LIN {X 0,Y 590.51,Z 609.214,A -85,B 0,C 180,E1 25169.414,E2 25169.414} C_VEL
LIN {X 0,Y 592.528,Z 625.3,A -85,B 0,C 180,E1 25167.889,E2 25167.889} C_VEL
LIN {X 0,Y 596.332,Z 639.507,A -85,B 0,C 180,E1 25166.405,E2 25166.405} C_VEL
LIN {X 0,Y 601.555,Z 651.727,A -85,B 0,C 180,E1 25165.009,E2 25165.009} C_VEL
LIN {X 0,Y 609.366,Z 664.255,A -85,B 0,C 180,E1 25163.442,E2 25163.442} C_VEL
LIN {X 0,Y 618.653,Z 674.701,A -85,B 0,C 180,E1 25161.991,E2 25161.991} C_VEL
LIN {X 0,Y 629.151,Z 683.449,A -85,B 0,C 180,E1 25160.645,E2 25160.645} C_VEL
LIN {X 0,Y 642.075,Z 691.353,A -85,B 0,C 180,E1 25159.269,E2 25159.269} C_VEL
LIN {X 0,Y 642.773,Z 691.86,A -85,B 0,C 180,E1 25159.192,E2 25159.192} C_VEL
LIN {X 0,Y 632.79,Z 705.423,A -85,B 0,C 180,E1 25158.911,E2 25158.911} C_VEL
LIN {X 0,Y 627.199,Z 713.768,A -85,B 0,C 180,E1 25158.699,E2 25158.699} C_VEL
LIN {X 0,Y 617.726,Z 726.944,A -85,B 0,C 180,E1 25158.399,E2 25158.399} C_VEL
LIN {X 0,Y 610.205,Z 739.734,A -85,B 0,C 180,E1 25157.994,E2 25157.994} C_VEL
LIN {X 0,Y 606.308,Z 747.166,A -85,B 0,C 180,E1 25157.757,E2 25157.757} C_VEL
LIN {X 0,Y 604.005,Z 763.89,A -85,B 0,C 180,E1 25157.714,E2 25157.714} C_VEL
LIN {X 0,Y 603.207,Z 776.285,A -85,B 0,C 180,E1 25157.587,E2 25157.587} C_VEL
LIN {X 0,Y 601.713,Z 819.453,A -85,B 0,C 180,E1 25156.959,E2 25156.959} C_VEL
LIN {X 0,Y 599.605,Z 849.263,A -85,B 0,C 180,E1 25156.4,E2 25156.4} C_VEL
LIN {X 0,Y 597.26,Z 876.114,A -85,B 0,C 180,E1 25155.731,E2 25155.731} C_VEL
LIN {X 0,Y 594.587,Z 902.786,A -85,B 0,C 180,E1 25154.898,E2 25154.898} C_VEL
LIN {X 0,Y 591.585,Z 928.736,A -85,B 0,C 180,E1 25153.901,E2 25153.901} C_VEL
LIN {X 0,Y 588.504,Z 952.603,A -85,B 0,C 180,E1 25152.811,E2 25152.811} C_VEL
LIN {X 0,Y 584.931,Z 977.211,A -85,B 0,C 180,E1 25151.481,E2 25151.481} C_VEL
LIN {X 0,Y 581.177,Z 1000.865,A -85,B 0,C 180,E1 25149.983,E2 25149.983} C_VEL
LIN {X 0,Y 577.362,Z 1023.647,A -85,B 0,C 180,E1 25148.313,E2 25148.313} C_VEL
LIN {X 0,Y 573.393,Z 1045.93,A -85,B 0,C 180,E1 25146.423,E2 25146.423} C_VEL
LIN {X 0,Y 569.931,Z 1065.063,A -85,B 0,C 180,E1 25144.577,E2 25144.577} C_VEL
LIN {X 0,Y 566.236,Z 1085.757,A -85,B 0,C 180,E1 25142.312,E2 25142.312} C_VEL
LIN {X 0,Y 563.29,Z 1102.922,A -85,B 0,C 180,E1 25140.177,E2 25140.177} C_VEL
LIN {X 0,Y 560.401,Z 1120.145,A -85,B 0,C 180,E1 25137.75,E2 25137.75} C_VEL
LIN {X 0,Y 558.227,Z 1134.517,A -85,B 0,C 180,E1 25135.458,E2 25135.458} C_VEL
LIN {X 0,Y 556.22,Z 1148.88,A -85,B 0,C 180,E1 25132.847,E2 25132.847} C_VEL
LIN {X 0,Y 554.619,Z 1162.074,A -85,B 0,C 180,E1 25130.068,E2 25130.068} C_VEL
LIN {X 0,Y 553.529,Z 1172.793,A -85,B 0,C 180,E1 25127.448,E2 25127.448} C_VEL
LIN {X 0,Y 552.746,Z 1182.624,A -85,B 0,C 180,E1 25124.581,E2 25124.581} C_VEL
LIN {X 0,Y 552.293,Z 1190.071,A -85,B 0,C 180,E1 25121.909,E2 25121.909} C_VEL
LIN {X 0,Y 552.049,Z 1196.15,A -85,B 0,C 180,E1 25119.17,E2 25119.17} C_VEL
LIN {X 0,Y 551.953,Z 1200.501,A -85,B 0,C 180,E1 25116.552,E2 25116.552} C_VEL
LIN {X 0,Y 551.914,Z 1203.328,A -85,B 0,C 180,E1 25113.946,E2 25113.946} C_VEL
LIN {X 0,Y 551.916,Z 1204.787,A -85,B 0,C 180,E1 25111.244,E2 25111.244} C_VEL
LIN {X 0,Y 551.916,Z 1204.786,A -85,B 0,C 180,E1 25108.753,E2 25108.753} C_VEL
LIN {X 0,Y 551.914,Z 1203.326,A -85,B 0,C 180,E1 25106.051,E2 25106.051} C_VEL
LIN {X 0,Y 551.951,Z 1200.497,A -85,B 0,C 180,E1 25103.445,E2 25103.445} C_VEL
LIN {X 0,Y 552.051,Z 1196.087,A -85,B 0,C 180,E1 25100.796,E2 25100.796} C_VEL
LIN {X 0,Y 552.293,Z 1190.065,A -85,B 0,C 180,E1 25098.088,E2 25098.088} C_VEL
LIN {X 0,Y 552.746,Z 1182.623,A -85,B 0,C 180,E1 25095.419,E2 25095.419} C_VEL
LIN {X 0,Y 553.529,Z 1172.783,A -85,B 0,C 180,E1 25092.55,E2 25092.55} C_VEL
LIN {X 0,Y 554.62,Z 1162.073,A -85,B 0,C 180,E1 25089.932,E2 25089.932} C_VEL
LIN {X 0,Y 556.222,Z 1148.866,A -85,B 0,C 180,E1 25087.151,E2 25087.151} C_VEL
LIN {X 0,Y 558.249,Z 1134.381,A -85,B 0,C 180,E1 25084.519,E2 25084.519} C_VEL
LIN {X 0,Y 560.406,Z 1120.11,A -85,B 0,C 180,E1 25082.245,E2 25082.245} C_VEL
LIN {X 0,Y 563.403,Z 1102.225,A -85,B 0,C 180,E1 25079.733,E2 25079.733} C_VEL
LIN {X 0,Y 566.285,Z 1085.478,A -85,B 0,C 180,E1 25077.655,E2 25077.655} C_VEL
LIN {X 0,Y 569.935,Z 1065.037,A -85,B 0,C 180,E1 25075.42,E2 25075.42} C_VEL
LIN {X 0,Y 573.399,Z 1045.901,A -85,B 0,C 180,E1 25073.575,E2 25073.575} C_VEL
LIN {X 0,Y 577.128,Z 1024.944,A -85,B 0,C 180,E1 25071.792,E2 25071.792} C_VEL
LIN {X 0,Y 580.932,Z 1002.513,A -85,B 0,C 180,E1 25070.129,E2 25070.129} C_VEL
LIN {X 0,Y 584.659,Z 978.962,A -85,B 0,C 180,E1 25068.623,E2 25068.623} C_VEL
LIN {X 0,Y 588.218,Z 954.716,A -85,B 0,C 180,E1 25067.293,E2 25067.293} C_VEL
LIN {X 0,Y 591.704,Z 928.188,A -85,B 0,C 180,E1 25066.07,E2 25066.07} C_VEL
LIN {X 0,Y 594.755,Z 901.513,A -85,B 0,C 180,E1 25065.055,E2 25065.055} C_VEL
LIN {X 0,Y 597.525,Z 873.698,A -85,B 0,C 180,E1 25064.197,E2 25064.197} C_VEL
LIN {X 0,Y 600.006,Z 844.404,A -85,B 0,C 180,E1 25063.494,E2 25063.494} C_VEL
LIN {X 0,Y 602.162,Z 810.979,A -85,B 0,C 180,E1 25062.904,E2 25062.904} C_VEL
LIN {X 0,Y 604.764,Z 734.901,A -85,B 0,C 180,E1 25061.837,E2 25061.837} C_VEL
LIN {X 0,Y 611.43,Z 660.897,A -85,B 0,C 180,E1 25060.584,E2 25060.584} C_VEL
LIN {X 0,Y 612.883,Z 645.219,A -85,B 0,C 180,E1 25060.323,E2 25060.323} C_VEL
LIN {X 0,Y 616.334,Z 610.333,A -85,B 0,C 180,E1 25059.764,E2 25059.764} C_VEL
LIN {X 0,Y 617.889,Z 595.942,A -85,B 0,C 180,E1 25059.548,E2 25059.548} C_VEL
LIN {X 0,Y 620.532,Z 567.007,A -85,B 0,C 180,E1 25059.061,E2 25059.061} C_VEL
LIN {X 0,Y 624,Z 538.188,A -85,B 0,C 180,E1 25058.666,E2 25058.666} C_VEL
LIN {X 0,Y 626.222,Z 512.687,A -85,B 0,C 180,E1 25058.225,E2 25058.225} C_VEL
LIN {X 0,Y 630.739,Z 478.238,A -85,B 0,C 180,E1 25057.795,E2 25057.795} C_VEL
LIN {X 0,Y 632.724,Z 453.547,A -85,B 0,C 180,E1 25057.35,E2 25057.35} C_VEL
LIN {X 0,Y 633.686,Z 444.389,A -85,B 0,C 180,E1 25057.21,E2 25057.21} C_VEL
LIN {X 0,Y 625.904,Z 434.82,A -85,B 0,C 180,E1 25056.064,E2 25056.064} C_VEL
LIN {X 0,Y 610.871,Z 411.674,A -85,B 0,C 180,E1 25053.534,E2 25053.534} C_VEL
LIN {X 0,Y 599.2,Z 394.973,A -85,B 0,C 180,E1 25051.403,E2 25051.403} C_VEL
LIN {X 0,Y 589.319,Z 381.338,A -85,B 0,C 180,E1 25049.447,E2 25049.447} C_VEL
LIN {X 0,Y 584.227,Z 374.732,A -85,B 0,C 180,E1 25048.383,E2 25048.383} C_VEL
LIN {X 0,Y 581.035,Z 370.541,A -85,B 0,C 180,E1 25047.687,E2 25047.687} C_VEL
LIN {X 0,Y 576.918,Z 365.165,A -85,B 0,C 180,E1 25046.756,E2 25046.756} C_VEL
LIN {X 0,Y 573.423,Z 360.486,A -85,B 0,C 180,E1 25045.928,E2 25045.928} C_VEL
LIN {X 0,Y 569.377,Z 355.739,A -85,B 0,C 180,E1 25044.955,E2 25044.955} C_VEL
LIN {X 0,Y 568.216,Z 353.937,A -85,B 0,C 180,E1 25044.649,E2 25044.649} C_VEL
LIN {X 0,Y 565.016,Z 350.609,A -85,B 0,C 180,E1 25043.852,E2 25043.852} C_VEL
LIN {X 0,Y 563.518,Z 347.975,A -85,B 0,C 180,E1 25043.42,E2 25043.42} C_VEL
LIN {X 0,Y 560.374,Z 345.311,A -85,B 0,C 180,E1 25042.614,E2 25042.614} C_VEL
LIN {X 0,Y 558.326,Z 341.668,A -85,B 0,C 180,E1 25041.981,E2 25041.981} C_VEL
LIN {X 0,Y 555.306,Z 339.437,A -85,B 0,C 180,E1 25041.163,E2 25041.163} C_VEL
LIN {X 0,Y 553.735,Z 336.439,A -85,B 0,C 180,E1 25040.631,E2 25040.631} C_VEL
LIN {X 0,Y 553.497,Z 335.263,A -85,B 0,C 180,E1 25040.488,E2 25040.488} C_VEL
LIN {X 0,Y 553.496,Z 335.262,A -85,B 0,C 180,E1 25037.017,E2 25037.017} C_VEL
LIN {X 0,Y 553.524,Z 335.519,A -85,B 0,C 180,E1 25035.601,E2 25035.601} C_VEL
LIN {X 0,Y 560.446,Z 355.632,A -85,B 0,C 180,E1 25034.584,E2 25034.584} C_VEL
LIN {X 0,Y 560.203,Z 434.439,A -85,B 0,C 180,E1 25031.766,E2 25031.766} C_VEL
LIN {X 0,Y 560.354,Z 519.456,A -85,B 0,C 180,E1 25028.569,E2 25028.569} C_VEL
LIN {X 0,Y 560.071,Z 596.427,A -85,B 0,C 180,E1 25025.584,E2 25025.584} C_VEL
LIN {X 0,Y 559.404,Z 672.282,A -85,B 0,C 180,E1 25022.561,E2 25022.561} C_VEL
LIN {X 0,Y 558.433,Z 749.146,A -85,B 0,C 180,E1 25019.436,E2 25019.436} C_VEL
LIN {X 0,Y 557.327,Z 828.653,A -85,B 0,C 180,E1 25016.142,E2 25016.142} C_VEL
LIN {X 0,Y 556.701,Z 851.757,A -85,B 0,C 180,E1 25015.186,E2 25015.186} C_VEL
LIN {X 0,Y 556.119,Z 860.24,A -85,B 0,C 180,E1 25014.87,E2 25014.87} C_VEL
LIN {X 0,Y 555.338,Z 973.856,A -85,B 0,C 180,E1 25013.286,E2 25013.286} C_VEL
LIN {X 0,Y 555.38,Z 986.399,A -85,B 0,C 180,E1 25012.978,E2 25012.978} C_VEL
LIN {X 0,Y 555.343,Z 998.353,A -85,B 0,C 180,E1 25012.551,E2 25012.551} C_VEL
LIN {X 0,Y 555.203,Z 1011.407,A -85,B 0,C 180,E1 25011.925,E2 25011.925} C_VEL
LIN {X 0,Y 554.96,Z 1023.564,A -85,B 0,C 180,E1 25011.132,E2 25011.132} C_VEL
LIN {X 0,Y 554.721,Z 1033.15,A -85,B 0,C 180,E1 25010.35,E2 25010.35} C_VEL
LIN {X 0,Y 554.462,Z 1041.636,A -85,B 0,C 180,E1 25009.506,E2 25009.506} C_VEL
LIN {X 0,Y 554.197,Z 1049.49,A -85,B 0,C 180,E1 25008.553,E2 25008.553} C_VEL
LIN {X 0,Y 553.925,Z 1057.258,A -85,B 0,C 180,E1 25007.384,E2 25007.384} C_VEL
LIN {X 0,Y 553.645,Z 1064.108,A -85,B 0,C 180,E1 25005.995,E2 25005.995} C_VEL
LIN {X 0,Y 553.48,Z 1068.39,A -85,B 0,C 180,E1 25004.814,E2 25004.814} C_VEL
LIN {X 0,Y 553.352,Z 1071.423,A -85,B 0,C 180,E1 25003.627,E2 25003.627} C_VEL
LIN {X 0,Y 553.276,Z 1073.272,A -85,B 0,C 180,E1 25002.434,E2 25002.434} C_VEL
LIN {X 0,Y 553.227,Z 1074.038,A -85,B 0,C 180,E1 25001.014,E2 25001.014} C_VEL
LIN {X 0,Y 553.232,Z 1072.866,A -85,B 0,C 180,E1 24999.426,E2 24999.426} C_VEL
LIN {X 0,Y 553.274,Z 1070.476,A -85,B 0,C 180,E1 24998.143,E2 24998.143} C_VEL
LIN {X 0,Y 553.376,Z 1066.816,A -85,B 0,C 180,E1 24996.884,E2 24996.884} C_VEL
LIN {X 0,Y 553.578,Z 1060.937,A -85,B 0,C 180,E1 24995.453,E2 24995.453} C_VEL
LIN {X 0,Y 553.81,Z 1053.905,A -85,B 0,C 180,E1 24994.207,E2 24994.207} C_VEL
LIN {X 0,Y 554.066,Z 1046.433,A -85,B 0,C 180,E1 24993.151,E2 24993.151} C_VEL
LIN {X 0,Y 554.352,Z 1037.727,A -85,B 0,C 180,E1 24992.15,E2 24992.15} C_VEL
LIN {X 0,Y 554.704,Z 1026.532,A -85,B 0,C 180,E1 24991.113,E2 24991.113} C_VEL
LIN {X 0,Y 554.983,Z 1014.283,A -85,B 0,C 180,E1 24990.241,E2 24990.241} C_VEL
LIN {X 0,Y 555.2,Z 1003.236,A -85,B 0,C 180,E1 24989.617,E2 24989.617} C_VEL
LIN {X 0,Y 555.368,Z 990.76,A -85,B 0,C 180,E1 24989.071,E2 24989.071} C_VEL
LIN {X 0,Y 555.439,Z 974.896,A -85,B 0,C 180,E1 24988.598,E2 24988.598} C_VEL
LIN {X 0,Y 555.398,Z 958.822,A -85,B 0,C 180,E1 24988.323,E2 24988.323} C_VEL
LIN {X 0,Y 556.342,Z 853.596,A -85,B 0,C 180,E1 24986.88,E2 24986.88} C_VEL
LIN {X 0,Y 557.037,Z 837.818,A -85,B 0,C 180,E1 24986.212,E2 24986.212} C_VEL
LIN {X 0,Y 558.557,Z 756.681,A -85,B 0,C 180,E1 24982.702,E2 24982.702} C_VEL
LIN {X 0,Y 558.996,Z 735.045,A -85,B 0,C 180,E1 24981.765,E2 24981.765} C_VEL
LIN {X 0,Y 559.725,Z 732.326,A -85,B 0,C 180,E1 24981.556,E2 24981.556} C_VEL
LIN {X 0,Y 561.703,Z 730.328,A -85,B 0,C 180,E1 24981.216,E2 24981.216} C_VEL
LIN {X 0,Y 566.453,Z 728.934,A -85,B 0,C 180,E1 24980.588,E2 24980.588} C_VEL
LIN {X 0,Y 571.435,Z 727.549,A -85,B 0,C 180,E1 24980.042,E2 24980.042} C_VEL
LIN {X 0,Y 572.537,Z 726.951,A -85,B 0,C 180,E1 24979.933,E2 24979.933} C_VEL
LIN {X 0,Y 577.099,Z 723.151,A -85,B 0,C 180,E1 24979.527,E2 24979.527} C_VEL
LIN {X 0,Y 582.053,Z 717.036,A -85,B 0,C 180,E1 24979.15,E2 24979.15} C_VEL
LIN {X 0,Y 587.21,Z 712.981,A -85,B 0,C 180,E1 24978.713,E2 24978.713} C_VEL
LIN {X 0,Y 593.112,Z 706.301,A -85,B 0,C 180,E1 24978.28,E2 24978.28} C_VEL
LIN {X 0,Y 594.096,Z 705.686,A -85,B 0,C 180,E1 24978.198,E2 24978.198} C_VEL
LIN {X 0,Y 589.64,Z 797.135,A -85,B 0,C 180,E1 24976.661,E2 24976.661} C_VEL
LIN {X 0,Y 588.016,Z 826.067,A -85,B 0,C 180,E1 24976.11,E2 24976.11} C_VEL
LIN {X 0,Y 585.936,Z 855.454,A -85,B 0,C 180,E1 24975.37,E2 24975.37} C_VEL
LIN {X 0,Y 583.804,Z 880.901,A -85,B 0,C 180,E1 24974.562,E2 24974.562} C_VEL
LIN {X 0,Y 581.521,Z 904.72,A -85,B 0,C 180,E1 24973.659,E2 24973.659} C_VEL
LIN {X 0,Y 578.69,Z 930.131,A -85,B 0,C 180,E1 24972.501,E2 24972.501} C_VEL
LIN {X 0,Y 575.93,Z 952.54,A -85,B 0,C 180,E1 24971.317,E2 24971.317} C_VEL
LIN {X 0,Y 572.684,Z 976.437,A -85,B 0,C 180,E1 24969.85,E2 24969.85} C_VEL
LIN {X 0,Y 568.97,Z 1000.766,A -85,B 0,C 180,E1 24968.086,E2 24968.086} C_VEL
LIN {X 0,Y 565.934,Z 1019.321,A -85,B 0,C 180,E1 24966.543,E2 24966.543} C_VEL
LIN {X 0,Y 563.293,Z 1033.801,A -85,B 0,C 180,E1 24965.142,E2 24965.142} C_VEL
LIN {X 0,Y 560.146,Z 1050.417,A -85,B 0,C 180,E1 24963.342,E2 24963.342} C_VEL
LIN {X 0,Y 557.391,Z 1065.236,A -85,B 0,C 180,E1 24961.56,E2 24961.56} C_VEL
LIN {X 0,Y 554.87,Z 1079.174,A -85,B 0,C 180,E1 24959.706,E2 24959.706} C_VEL
LIN {X 0,Y 552.605,Z 1092.304,A -85,B 0,C 180,E1 24957.772,E2 24957.772} C_VEL
LIN {X 0,Y 550.606,Z 1104.824,A -85,B 0,C 180,E1 24955.724,E2 24955.724} C_VEL
LIN {X 0,Y 548.637,Z 1118.142,A -85,B 0,C 180,E1 24953.286,E2 24953.286} C_VEL
LIN {X 0,Y 546.891,Z 1131.542,A -85,B 0,C 180,E1 24950.44,E2 24950.44} C_VEL
LIN {X 0,Y 545.8,Z 1141.259,A -85,B 0,C 180,E1 24948.048,E2 24948.048} C_VEL
LIN {X 0,Y 545.07,Z 1148.997,A -85,B 0,C 180,E1 24945.864,E2 24945.864} C_VEL
LIN {X 0,Y 544.565,Z 1155.927,A -85,B 0,C 180,E1 24943.594,E2 24943.594} C_VEL
LIN {X 0,Y 544.215,Z 1161.96,A -85,B 0,C 180,E1 24941.232,E2 24941.232} C_VEL
LIN {X 0,Y 544.045,Z 1166.607,A -85,B 0,C 180,E1 24938.989,E2 24938.989} C_VEL
LIN {X 0,Y 543.953,Z 1170.204,A -85,B 0,C 180,E1 24936.757,E2 24936.757} C_VEL
LIN {X 0,Y 543.916,Z 1172.778,A -85,B 0,C 180,E1 24934.535,E2 24934.535} C_VEL
LIN {X 0,Y 543.908,Z 1174.344,A -85,B 0,C 180,E1 24932.319,E2 24932.319} C_VEL
LIN {X 0,Y 543.907,Z 1174.912,A -85,B 0,C 180,E1 24929.896,E2 24929.896} C_VEL
LIN {X 0,Y 543.907,Z 1174.289,A -85,B 0,C 180,E1 24927.473,E2 24927.473} C_VEL
LIN {X 0,Y 543.92,Z 1172.538,A -85,B 0,C 180,E1 24925.114,E2 24925.114} C_VEL
LIN {X 0,Y 543.973,Z 1169.598,A -85,B 0,C 180,E1 24922.715,E2 24922.715} C_VEL
LIN {X 0,Y 544.113,Z 1164.806,A -85,B 0,C 180,E1 24919.947,E2 24919.947} C_VEL
LIN {X 0,Y 544.467,Z 1157.685,A -85,B 0,C 180,E1 24916.947,E2 24916.947} C_VEL
LIN {X 0,Y 544.968,Z 1150.356,A -85,B 0,C 180,E1 24914.464,E2 24914.464} C_VEL
LIN {X 0,Y 545.68,Z 1142.458,A -85,B 0,C 180,E1 24912.183,E2 24912.183} C_VEL
LIN {X 0,Y 546.618,Z 1133.78,A -85,B 0,C 180,E1 24909.999,E2 24909.999} C_VEL
LIN {X 0,Y 547.759,Z 1124.416,A -85,B 0,C 180,E1 24907.913,E2 24907.913} C_VEL
LIN {X 0,Y 549.227,Z 1113.891,A -85,B 0,C 180,E1 24905.821,E2 24905.821} C_VEL
LIN {X 0,Y 551.035,Z 1101.917,A -85,B 0,C 180,E1 24903.689,E2 24903.689} C_VEL
LIN {X 0,Y 553.601,Z 1086.776,A -85,B 0,C 180,E1 24901.288,E2 24901.288} C_VEL
LIN {X 0,Y 556.821,Z 1068.311,A -85,B 0,C 180,E1 24898.739,E2 24898.739} C_VEL
LIN {X 0,Y 559.75,Z 1052.486,A -85,B 0,C 180,E1 24896.806,E2 24896.806} C_VEL
LIN {X 0,Y 562.67,Z 1036.971,A -85,B 0,C 180,E1 24895.098,E2 24895.098} C_VEL
LIN {X 0,Y 565.344,Z 1022.647,A -85,B 0,C 180,E1 24893.668,E2 24893.668} C_VEL
LIN {X 0,Y 567.988,Z 1006.559,A -85,B 0,C 180,E1 24892.287,E2 24892.287} C_VEL
LIN {X 0,Y 571.311,Z 985.32,A -85,B 0,C 180,E1 24890.676,E2 24890.676} C_VEL
LIN {X 0,Y 574.184,Z 965.577,A -85,B 0,C 180,E1 24889.364,E2 24889.364} C_VEL
LIN {X 0,Y 576.941,Z 944.473,A -85,B 0,C 180,E1 24888.148,E2 24888.148} C_VEL
LIN {X 0,Y 579.829,Z 920.099,A -85,B 0,C 180,E1 24886.933,E2 24886.933} C_VEL
LIN {X 0,Y 582.213,Z 897.637,A -85,B 0,C 180,E1 24885.969,E2 24885.969} C_VEL
LIN {X 0,Y 584.057,Z 877.701,A -85,B 0,C 180,E1 24885.242,E2 24885.242} C_VEL
LIN {X 0,Y 586.31,Z 850.909,A -85,B 0,C 180,E1 24884.413,E2 24884.413} C_VEL
LIN {X 0,Y 587.914,Z 826.678,A -85,B 0,C 180,E1 24883.823,E2 24883.823} C_VEL
LIN {X 0,Y 589.099,Z 806.755,A -85,B 0,C 180,E1 24883.424,E2 24883.424} C_VEL
LIN {X 0,Y 595.542,Z 680.019,A -85,B 0,C 180,E1 24881.271,E2 24881.271} C_VEL
LIN {X 0,Y 603.788,Z 534.875,A -85,B 0,C 180,E1 24878.84,E2 24878.84} C_VEL
LIN {X 0,Y 608.499,Z 434.897,A -85,B 0,C 180,E1 24877.284,E2 24877.284} C_VEL
LIN {X 0,Y 608.958,Z 420.597,A -85,B 0,C 180,E1 24877.057,E2 24877.057} C_VEL
LIN {X 0,Y 597.614,Z 409.55,A -85,B 0,C 180,E1 24875.344,E2 24875.344} C_VEL
LIN {X 0,Y 588.958,Z 401.686,A -85,B 0,C 180,E1 24873.956,E2 24873.956} C_VEL
LIN {X 0,Y 582.445,Z 395.957,A -85,B 0,C 180,E1 24872.853,E2 24872.853} C_VEL
LIN {X 0,Y 579.818,Z 393.63,A -85,B 0,C 180,E1 24872.369,E2 24872.369} C_VEL
LIN {X 0,Y 578.408,Z 390.814,A -85,B 0,C 180,E1 24871.355,E2 24871.355} C_VEL
LIN {X 0,Y 575.887,Z 386.066,A -85,B 0,C 180,E1 24869.43,E2 24869.43} C_VEL
LIN {X 0,Y 573.641,Z 381.867,A -85,B 0,C 180,E1 24867.479,E2 24867.479} C_VEL
LIN {X 0,Y 570.817,Z 376.935,A -85,B 0,C 180,E1 24864.621,E2 24864.621} C_VEL
LIN {X 0,Y 570.206,Z 375.881,A -85,B 0,C 180,E1 24863.896,E2 24863.896} C_VEL
LIN {X 0,Y 567.555,Z 370.875,A -85,B 0,C 180,E1 24859.449,E2 24859.449} C_VEL
LIN {X 0,Y 566.073,Z 369.458,A -85,B 0,C 180,E1 24854.84,E2 24854.84} C_VEL
LIN {X 0,Y 566.639,Z 370.081,A -85,B 0,C 180,E1 24850.781,E2 24850.781} C_VEL
LIN {X 0,Y 567.835,Z 371.39,A -85,B 0,C 180,E1 24848.28,E2 24848.28} C_VEL
LIN {X 0,Y 570.94,Z 376.86,A -85,B 0,C 180,E1 24843.715,E2 24843.715} C_VEL
LIN {X 0,Y 573.241,Z 381.117,A -85,B 0,C 180,E1 24841.299,E2 24841.299} C_VEL
LIN {X 0,Y 573.954,Z 382.347,A -85,B 0,C 180,E1 24840.664,E2 24840.664} C_VEL
LIN {X 0,Y 576.229,Z 386.32,A -85,B 0,C 180,E1 24838.807,E2 24838.807} C_VEL
LIN {X 0,Y 579.608,Z 392.611,A -85,B 0,C 180,E1 24836.34,E2 24836.34} C_VEL
LIN {X 0,Y 582.344,Z 397.71,A -85,B 0,C 180,E1 24834.581,E2 24834.581} C_VEL
LIN {X 0,Y 584.961,Z 402.676,A -85,B 0,C 180,E1 24833.029,E2 24833.029} C_VEL
LIN {X 0,Y 587.586,Z 407.673,A -85,B 0,C 180,E1 24831.585,E2 24831.585} C_VEL
LIN {X 0,Y 591.706,Z 415.65,A -85,B 0,C 180,E1 24829.484,E2 24829.484} C_VEL
LIN {X 0,Y 597.53,Z 427.473,A -85,B 0,C 180,E1 24826.747,E2 24826.747} C_VEL
LIN {X 0,Y 603.495,Z 440.421,A -85,B 0,C 180,E1 24824.135,E2 24824.135} C_VEL
LIN {X 0,Y 604.72,Z 443.335,A -85,B 0,C 180,E1 24823.601,E2 24823.601} C_VEL
LIN {X 0,Y 599.356,Z 478.045,A -85,B 0,C 180,E1 24820.61,E2 24820.61} C_VEL
LIN {X 0,Y 594.302,Z 512.72,A -85,B 0,C 180,E1 24817.756,E2 24817.756} C_VEL
LIN {X 0,Y 589.378,Z 549.232,A -85,B 0,C 180,E1 24814.851,E2 24814.851} C_VEL
LIN {X 0,Y 584.185,Z 594.684,A -85,B 0,C 180,E1 24811.308,E2 24811.308} C_VEL
LIN {X 0,Y 584.176,Z 612.88,A -85,B 0,C 180,E1 24809.73,E2 24809.73} C_VEL
LIN {X 0,Y 586.102,Z 628.98,A -85,B 0,C 180,E1 24808.186,E2 24808.186} C_VEL
LIN {X 0,Y 589.787,Z 643.265,A -85,B 0,C 180,E1 24806.681,E2 24806.681} C_VEL
LIN {X 0,Y 594.874,Z 655.617,A -85,B 0,C 180,E1 24805.263,E2 24805.263} C_VEL
LIN {X 0,Y 602.522,Z 668.326,A -85,B 0,C 180,E1 24803.669,E2 24803.669} C_VEL
LIN {X 0,Y 611.632,Z 679.01,A -85,B 0,C 180,E1 24802.19,E2 24802.19} C_VEL
LIN {X 0,Y 622.56,Z 688.475,A -85,B 0,C 180,E1 24800.743,E2 24800.743} C_VEL
LIN {X 0,Y 632.882,Z 695.437,A -85,B 0,C 180,E1 24799.579,E2 24799.579} C_VEL
LIN {X 0,Y 624.075,Z 708.29,A -85,B 0,C 180,E1 24799.271,E2 24799.271} C_VEL
LIN {X 0,Y 612.294,Z 724.665,A -85,B 0,C 180,E1 24798.904,E2 24798.904} C_VEL
LIN {X 0,Y 604.358,Z 738.022,A -85,B 0,C 180,E1 24798.486,E2 24798.486} C_VEL
LIN {X 0,Y 601.573,Z 743.536,A -85,B 0,C 180,E1 24798.316,E2 24798.316} C_VEL
LIN {X 0,Y 599.265,Z 758.516,A -85,B 0,C 180,E1 24798.304,E2 24798.304} C_VEL
LIN {X 0,Y 597.904,Z 773.102,A -85,B 0,C 180,E1 24798.198,E2 24798.198} C_VEL
LIN {X 0,Y 596.316,Z 817.198,A -85,B 0,C 180,E1 24797.553,E2 24797.553} C_VEL
LIN {X 0,Y 594.025,Z 848.758,A -85,B 0,C 180,E1 24796.963,E2 24796.963} C_VEL
LIN {X 0,Y 591.422,Z 877.702,A -85,B 0,C 180,E1 24796.238,E2 24796.238} C_VEL
LIN {X 0,Y 588.576,Z 904.677,A -85,B 0,C 180,E1 24795.38,E2 24795.38} C_VEL
LIN {X 0,Y 585.764,Z 927.976,A -85,B 0,C 180,E1 24794.478,E2 24794.478} C_VEL
LIN {X 0,Y 582.666,Z 951.398,A -85,B 0,C 180,E1 24793.413,E2 24793.413} C_VEL
LIN {X 0,Y 579.101,Z 975.478,A -85,B 0,C 180,E1 24792.126,E2 24792.126} C_VEL
LIN {X 0,Y 575.44,Z 997.395,A -85,B 0,C 180,E1 24790.747,E2 24790.747} C_VEL
LIN {X 0,Y 571.21,Z 1021.62,A -85,B 0,C 180,E1 24788.994,E2 24788.994} C_VEL
LIN {X 0,Y 567.046,Z 1044.191,A -85,B 0,C 180,E1 24787.087,E2 24787.087} C_VEL
LIN {X 0,Y 563.262,Z 1063.982,A -85,B 0,C 180,E1 24785.171,E2 24785.171} C_VEL
LIN {X 0,Y 559.56,Z 1083.663,A -85,B 0,C 180,E1 24783.023,E2 24783.023} C_VEL
LIN {X 0,Y 556.432,Z 1100.552,A -85,B 0,C 180,E1 24780.924,E2 24780.924} C_VEL
LIN {X 0,Y 553.386,Z 1117.974,A -85,B 0,C 180,E1 24778.488,E2 24778.488} C_VEL
LIN {X 0,Y 550.857,Z 1133.198,A -85,B 0,C 180,E1 24776.055,E2 24776.055} C_VEL
LIN {X 0,Y 548.685,Z 1147.76,A -85,B 0,C 180,E1 24773.406,E2 24773.406} C_VEL
LIN {X 0,Y 546.969,Z 1160.827,A -85,B 0,C 180,E1 24770.658,E2 24770.658} C_VEL
LIN {X 0,Y 545.788,Z 1171.565,A -85,B 0,C 180,E1 24768.034,E2 24768.034} C_VEL
LIN {X 0,Y 544.936,Z 1180.951,A -85,B 0,C 180,E1 24765.319,E2 24765.319} C_VEL
LIN {X 0,Y 544.375,Z 1188.99,A -85,B 0,C 180,E1 24762.516,E2 24762.516} C_VEL
LIN {X 0,Y 544.095,Z 1195.366,A -85,B 0,C 180,E1 24759.732,E2 24759.732} C_VEL
LIN {X 0,Y 543.965,Z 1199.881,A -85,B 0,C 180,E1 24757.073,E2 24757.073} C_VEL
LIN {X 0,Y 543.92,Z 1203.062,A -85,B 0,C 180,E1 24754.321,E2 24754.321} C_VEL
LIN {X 0,Y 543.908,Z 1204.699,A -85,B 0,C 180,E1 24751.684,E2 24751.684} C_VEL
LIN {X 0,Y 543.907,Z 1204.845,A -85,B 0,C 180,E1 24749.051,E2 24749.051} C_VEL
LIN {X 0,Y 543.913,Z 1203.677,A -85,B 0,C 180,E1 24746.415,E2 24746.415} C_VEL
LIN {X 0,Y 543.945,Z 1201.031,A -85,B 0,C 180,E1 24743.773,E2 24743.773} C_VEL
LIN {X 0,Y 544.038,Z 1196.928,A -85,B 0,C 180,E1 24741.118,E2 24741.118} C_VEL
LIN {X 0,Y 544.258,Z 1191.41,A -85,B 0,C 180,E1 24738.447,E2 24738.447} C_VEL
LIN {X 0,Y 544.712,Z 1183.952,A -85,B 0,C 180,E1 24735.651,E2 24735.651} C_VEL
LIN {X 0,Y 545.491,Z 1174.422,A -85,B 0,C 180,E1 24732.747,E2 24732.747} C_VEL
LIN {X 0,Y 546.638,Z 1163.636,A -85,B 0,C 180,E1 24729.997,E2 24729.997} C_VEL
LIN {X 0,Y 548.163,Z 1151.659,A -85,B 0,C 180,E1 24727.363,E2 24727.363} C_VEL
LIN {X 0,Y 550.326,Z 1136.805,A -85,B 0,C 180,E1 24724.556,E2 24724.556} C_VEL
LIN {X 0,Y 552.742,Z 1121.545,A -85,B 0,C 180,E1 24722.061,E2 24722.061} C_VEL
LIN {X 0,Y 555.728,Z 1104.764,A -85,B 0,C 180,E1 24719.629,E2 24719.629} C_VEL
LIN {X 0,Y 558.943,Z 1086.852,A -85,B 0,C 180,E1 24717.36,E2 24717.36} C_VEL
LIN {X 0,Y 562.586,Z 1067.591,A -85,B 0,C 180,E1 24715.197,E2 24715.197} C_VEL
LIN {X 0,Y 566.606,Z 1046.593,A -85,B 0,C 180,E1 24713.129,E2 24713.129} C_VEL
LIN {X 0,Y 570.212,Z 1027.155,A -85,B 0,C 180,E1 24711.452,E2 24711.452} C_VEL
LIN {X 0,Y 574.41,Z 1003.744,A -85,B 0,C 180,E1 24709.68,E2 24709.68} C_VEL
LIN {X 0,Y 578.265,Z 980.684,A -85,B 0,C 180,E1 24708.181,E2 24708.181} C_VEL
LIN {X 0,Y 582.05,Z 955.634,A -85,B 0,C 180,E1 24706.797,E2 24706.797} C_VEL
LIN {X 0,Y 585.496,Z 930.62,A -85,B 0,C 180,E1 24705.626,E2 24705.626} C_VEL
LIN {X 0,Y 588.686,Z 903.882,A -85,B 0,C 180,E1 24704.59,E2 24704.59} C_VEL
LIN {X 0,Y 591.584,Z 876.02,A -85,B 0,C 180,E1 24703.714,E2 24703.714} C_VEL
LIN {X 0,Y 594.182,Z 846.963,A -85,B 0,C 180,E1 24702.996,E2 24702.996} C_VEL
LIN {X 0,Y 596.465,Z 814.54,A -85,B 0,C 180,E1 24702.403,E2 24702.403} C_VEL
LIN {X 0,Y 598.405,Z 756.727,A -85,B 0,C 180,E1 24701.575,E2 24701.575} C_VEL
LIN {X 0,Y 599.593,Z 730.221,A -85,B 0,C 180,E1 24701.198,E2 24701.198} C_VEL
LIN {X 0,Y 606.118,Z 660.111,A -85,B 0,C 180,E1 24700.016,E2 24700.016} C_VEL
LIN {X 0,Y 607.72,Z 642.456,A -85,B 0,C 180,E1 24699.714,E2 24699.714} C_VEL
LIN {X 0,Y 611.474,Z 606.607,A -85,B 0,C 180,E1 24699.154,E2 24699.154} C_VEL
LIN {X 0,Y 612.598,Z 595.536,A -85,B 0,C 180,E1 24698.977,E2 24698.977} C_VEL
LIN {X 0,Y 615.456,Z 565.573,A -85,B 0,C 180,E1 24698.479,E2 24698.479} C_VEL
LIN {X 0,Y 618.733,Z 538.714,A -85,B 0,C 180,E1 24698.11,E2 24698.11} C_VEL
LIN {X 0,Y 621.076,Z 512.63,A -85,B 0,C 180,E1 24697.661,E2 24697.661} C_VEL
LIN {X 0,Y 625.775,Z 476.02,A -85,B 0,C 180,E1 24697.187,E2 24697.187} C_VEL
LIN {X 0,Y 627.695,Z 453.263,A -85,B 0,C 180,E1 24696.781,E2 24696.781} C_VEL
LIN {X 0,Y 628.114,Z 448.951,A -85,B 0,C 180,E1 24696.71,E2 24696.71} C_VEL
LIN {X 0,Y 620.495,Z 438.824,A -85,B 0,C 180,E1 24695.538,E2 24695.538} C_VEL
LIN {X 0,Y 607.119,Z 417.981,A -85,B 0,C 180,E1 24693.232,E2 24693.232} C_VEL
LIN {X 0,Y 594.255,Z 399.296,A -85,B 0,C 180,E1 24690.821,E2 24690.821} C_VEL
LIN {X 0,Y 582.659,Z 383.409,A -85,B 0,C 180,E1 24688.439,E2 24688.439} C_VEL
LIN {X 0,Y 573.839,Z 372.015,A -85,B 0,C 180,E1 24686.464,E2 24686.464} C_VEL
LIN {X 0,Y 569.498,Z 366.427,A -85,B 0,C 180,E1 24685.422,E2 24685.422} C_VEL
LIN {X 0,Y 566.058,Z 361.92,A -85,B 0,C 180,E1 24684.554,E2 24684.554} C_VEL
LIN {X 0,Y 561.848,Z 356.984,A -85,B 0,C 180,E1 24683.466,E2 24683.466} C_VEL
LIN {X 0,Y 560.565,Z 355.113,A -85,B 0,C 180,E1 24683.105,E2 24683.105} C_VEL
LIN {X 0,Y 557.356,Z 351.888,A -85,B 0,C 180,E1 24682.243,E2 24682.243} C_VEL
LIN {X 0,Y 555.801,Z 349.115,A -85,B 0,C 180,E1 24681.752,E2 24681.752} C_VEL
LIN {X 0,Y 552.685,Z 346.501,A -85,B 0,C 180,E1 24680.88,E2 24680.88} C_VEL
LIN {X 0,Y 550.89,Z 343.034,A -85,B 0,C 180,E1 24680.256,E2 24680.256} C_VEL
LIN {X 0,Y 547.191,Z 340.238,A -85,B 0,C 180,E1 24679.142,E2 24679.142} C_VEL
LIN {X 0,Y 545.756,Z 337.359,A -85,B 0,C 180,E1 24678.59,E2 24678.59} C_VEL
LIN {X 0,Y 545.554,Z 336.269,A -85,B 0,C 180,E1 24678.431,E2 24678.431} C_VEL
LIN {X 0,Y 545.577,Z 336.357,A -85,B 0,C 180,E1 24675.944,E2 24675.944} C_VEL
LIN {X 0,Y 553.078,Z 357.862,A -85,B 0,C 180,E1 24674.835,E2 24674.835} C_VEL
LIN {X 0,Y 552.712,Z 440.058,A -85,B 0,C 180,E1 24671.872,E2 24671.872} C_VEL
LIN {X 0,Y 552.819,Z 519.291,A -85,B 0,C 180,E1 24668.87,E2 24668.87} C_VEL
LIN {X 0,Y 552.549,Z 589.671,A -85,B 0,C 180,E1 24666.129,E2 24666.129} C_VEL
LIN {X 0,Y 551.952,Z 656.032,A -85,B 0,C 180,E1 24663.479,E2 24663.479} C_VEL
LIN {X 0,Y 550.945,Z 738.044,A -85,B 0,C 180,E1 24660.151,E2 24660.151} C_VEL
LIN {X 0,Y 549.757,Z 819.378,A -85,B 0,C 180,E1 24656.768,E2 24656.768} C_VEL
LIN {X 0,Y 549.038,Z 851.408,A -85,B 0,C 180,E1 24655.43,E2 24655.43} C_VEL
LIN {X 0,Y 548.335,Z 861.523,A -85,B 0,C 180,E1 24655.051,E2 24655.051} C_VEL
LIN {X 0,Y 547.511,Z 974.935,A -85,B 0,C 180,E1 24653.438,E2 24653.438} C_VEL
LIN {X 0,Y 547.557,Z 987.683,A -85,B 0,C 180,E1 24653.121,E2 24653.121} C_VEL
LIN {X 0,Y 547.522,Z 999.134,A -85,B 0,C 180,E1 24652.708,E2 24652.708} C_VEL
LIN {X 0,Y 547.379,Z 1012.3,A -85,B 0,C 180,E1 24652.073,E2 24652.073} C_VEL
LIN {X 0,Y 547.133,Z 1024.467,A -85,B 0,C 180,E1 24651.275,E2 24651.275} C_VEL
LIN {X 0,Y 546.875,Z 1034.291,A -85,B 0,C 180,E1 24650.465,E2 24650.465} C_VEL
LIN {X 0,Y 546.626,Z 1042.216,A -85,B 0,C 180,E1 24649.673,E2 24649.673} C_VEL
LIN {X 0,Y 546.369,Z 1049.556,A -85,B 0,C 180,E1 24648.79,E2 24648.79} C_VEL
LIN {X 0,Y 546.124,Z 1056.031,A -85,B 0,C 180,E1 24647.845,E2 24647.845} C_VEL
LIN {X 0,Y 545.883,Z 1062.022,A -85,B 0,C 180,E1 24646.764,E2 24646.764} C_VEL
LIN {X 0,Y 545.66,Z 1067.608,A -85,B 0,C 180,E1 24645.461,E2 24645.461} C_VEL
LIN {X 0,Y 545.464,Z 1071.997,A -85,B 0,C 180,E1 24643.931,E2 24643.931} C_VEL
LIN {X 0,Y 545.368,Z 1074.083,A -85,B 0,C 180,E1 24642.722,E2 24642.722} C_VEL
LIN {X 0,Y 545.311,Z 1075.016,A -85,B 0,C 180,E1 24641.505,E2 24641.505} C_VEL
LIN {X 0,Y 545.293,Z 1074.801,A -85,B 0,C 180,E1 24640.282,E2 24640.282} C_VEL
LIN {X 0,Y 545.307,Z 1073.425,A -85,B 0,C 180,E1 24639.05,E2 24639.05} C_VEL
LIN {X 0,Y 545.408,Z 1070.302,A -85,B 0,C 180,E1 24637.584,E2 24637.584} C_VEL
LIN {X 0,Y 545.556,Z 1065.136,A -85,B 0,C 180,E1 24636.106,E2 24636.106} C_VEL
LIN {X 0,Y 545.741,Z 1059.762,A -85,B 0,C 180,E1 24634.961,E2 24634.961} C_VEL
LIN {X 0,Y 545.987,Z 1052.951,A -85,B 0,C 180,E1 24633.814,E2 24633.814} C_VEL
LIN {X 0,Y 546.345,Z 1043.342,A -85,B 0,C 180,E1 24632.535,E2 24632.535} C_VEL
LIN {X 0,Y 546.676,Z 1033.118,A -85,B 0,C 180,E1 24631.485,E2 24631.485} C_VEL
LIN {X 0,Y 546.955,Z 1023.289,A -85,B 0,C 180,E1 24630.664,E2 24630.664} C_VEL
LIN {X 0,Y 547.211,Z 1012.899,A -85,B 0,C 180,E1 24629.956,E2 24629.956} C_VEL
LIN {X 0,Y 547.478,Z 999.675,A -85,B 0,C 180,E1 24629.244,E2 24629.244} C_VEL
LIN {X 0,Y 547.596,Z 985.368,A -85,B 0,C 180,E1 24628.703,E2 24628.703} C_VEL
LIN {X 0,Y 547.618,Z 973.05,A -85,B 0,C 180,E1 24628.381,E2 24628.381} C_VEL
LIN {X 0,Y 547.588,Z 950.661,A -85,B 0,C 180,E1 24628.037,E2 24628.037} C_VEL
LIN {X 0,Y 548.565,Z 854.558,A -85,B 0,C 180,E1 24626.695,E2 24626.695} C_VEL
LIN {X 0,Y 549.29,Z 839.558,A -85,B 0,C 180,E1 24626.056,E2 24626.056} C_VEL
LIN {X 0,Y 550.901,Z 757.642,A -85,B 0,C 180,E1 24622.483,E2 24622.483} C_VEL
LIN {X 0,Y 551.189,Z 745.761,A -85,B 0,C 180,E1 24621.951,E2 24621.951} C_VEL
LIN {X 0,Y 552.098,Z 747.081,A -85,B 0,C 180,E1 24621.794,E2 24621.794} C_VEL
LIN {X 0,Y 553.694,Z 747.025,A -85,B 0,C 180,E1 24621.595,E2 24621.595} C_VEL
LIN {X 0,Y 556.447,Z 744.575,A -85,B 0,C 180,E1 24621.327,E2 24621.327} C_VEL
LIN {X 0,Y 560.14,Z 738.791,A -85,B 0,C 180,E1 24621.047,E2 24621.047} C_VEL
LIN {X 0,Y 560.795,Z 737.904,A -85,B 0,C 180,E1 24620.994,E2 24620.994} C_VEL
LIN {X 0,Y 564.107,Z 736.291,A -85,B 0,C 180,E1 24620.645,E2 24620.645} C_VEL
LIN {X 0,Y 567.903,Z 732.414,A -85,B 0,C 180,E1 24620.312,E2 24620.312} C_VEL
LIN {X 0,Y 571.014,Z 727.769,A -85,B 0,C 180,E1 24620.084,E2 24620.084} C_VEL
LIN {X 0,Y 572.537,Z 726.951,A -85,B 0,C 180,E1 24619.933,E2 24619.933} C_VEL
LIN {X 0,Y 575.224,Z 726.33,A -85,B 0,C 180,E1 24619.651,E2 24619.651} C_VEL
LIN {X 0,Y 578.388,Z 727.613,A -85,B 0,C 180,E1 24619.276,E2 24619.276} C_VEL
LIN {X 0,Y 581.589,Z 731.048,A -85,B 0,C 180,E1 24618.854,E2 24618.854} C_VEL
LIN {X 0,Y 584.458,Z 737.002,A -85,B 0,C 180,E1 24618.414,E2 24618.414} C_VEL
LIN {X 0,Y 585.864,Z 743.056,A -85,B 0,C 180,E1 24618.128,E2 24618.128} C_VEL
LIN {X 0,Y 586.009,Z 747.445,A -85,B 0,C 180,E1 24618.01,E2 24618.01} C_VEL
LIN {X 0,Y 581.935,Z 817.657,A -85,B 0,C 180,E1 24616.735,E2 24616.735} C_VEL
LIN {X 0,Y 579.659,Z 848.353,A -85,B 0,C 180,E1 24615.978,E2 24615.978} C_VEL
LIN {X 0,Y 577.19,Z 877.386,A -85,B 0,C 180,E1 24615.084,E2 24615.084} C_VEL
LIN {X 0,Y 574.566,Z 904.119,A -85,B 0,C 180,E1 24614.075,E2 24614.075} C_VEL
LIN {X 0,Y 571.635,Z 930.564,A -85,B 0,C 180,E1 24612.878,E2 24612.878} C_VEL
LIN {X 0,Y 568.841,Z 952.488,A -85,B 0,C 180,E1 24611.707,E2 24611.707} C_VEL
LIN {X 0,Y 565.457,Z 977.156,A -85,B 0,C 180,E1 24610.19,E2 24610.19} C_VEL
LIN {X 0,Y 562.606,Z 995.933,A -85,B 0,C 180,E1 24608.857,E2 24608.857} C_VEL
LIN {X 0,Y 559.239,Z 1016.534,A -85,B 0,C 180,E1 24607.181,E2 24607.181} C_VEL
LIN {X 0,Y 556.005,Z 1035.223,A -85,B 0,C 180,E1 24605.447,E2 24605.447} C_VEL
LIN {X 0,Y 553.764,Z 1047.446,A -85,B 0,C 180,E1 24604.164,E2 24604.164} C_VEL
LIN {X 0,Y 550.52,Z 1063.964,A -85,B 0,C 180,E1 24602.179,E2 24602.179} C_VEL
LIN {X 0,Y 547.754,Z 1078.374,A -85,B 0,C 180,E1 24600.254,E2 24600.254} C_VEL
LIN {X 0,Y 545.379,Z 1091.237,A -85,B 0,C 180,E1 24598.35,E2 24598.35} C_VEL
LIN {X 0,Y 543.259,Z 1103.531,A -85,B 0,C 180,E1 24596.333,E2 24596.333} C_VEL
LIN {X 0,Y 541.408,Z 1115.171,A -85,B 0,C 180,E1 24594.206,E2 24594.206} C_VEL
LIN {X 0,Y 539.823,Z 1126.08,A -85,B 0,C 180,E1 24591.973,E2 24591.973} C_VEL
LIN {X 0,Y 538.326,Z 1138.024,A -85,B 0,C 180,E1 24589.195,E2 24589.195} C_VEL
LIN {X 0,Y 537.239,Z 1148.292,A -85,B 0,C 180,E1 24586.323,E2 24586.323} C_VEL
LIN {X 0,Y 536.662,Z 1155.325,A -85,B 0,C 180,E1 24584.018,E2 24584.018} C_VEL
LIN {X 0,Y 536.277,Z 1161.463,A -85,B 0,C 180,E1 24581.618,E2 24581.618} C_VEL
LIN {X 0,Y 536.072,Z 1166.212,A -85,B 0,C 180,E1 24579.34,E2 24579.34} C_VEL
LIN {X 0,Y 535.964,Z 1169.98,A -85,B 0,C 180,E1 24577.022,E2 24577.022} C_VEL
LIN {X 0,Y 535.918,Z 1172.678,A -85,B 0,C 180,E1 24574.71,E2 24574.71} C_VEL
LIN {X 0,Y 535.907,Z 1174.292,A -85,B 0,C 180,E1 24572.461,E2 24572.461} C_VEL
LIN {X 0,Y 535.906,Z 1174.908,A -85,B 0,C 180,E1 24570.108,E2 24570.108} C_VEL
LIN {X 0,Y 535.908,Z 1174.383,A -85,B 0,C 180,E1 24567.649,E2 24567.649} C_VEL
LIN {X 0,Y 535.916,Z 1172.86,A -85,B 0,C 180,E1 24565.4,E2 24565.4} C_VEL
LIN {X 0,Y 535.954,Z 1170.328,A -85,B 0,C 180,E1 24563.144,E2 24563.144} C_VEL
LIN {X 0,Y 536.05,Z 1166.774,A -85,B 0,C 180,E1 24560.879,E2 24560.879} C_VEL
LIN {X 0,Y 536.233,Z 1162.17,A -85,B 0,C 180,E1 24558.602,E2 24558.602} C_VEL
LIN {X 0,Y 536.584,Z 1156.479,A -85,B 0,C 180,E1 24556.312,E2 24556.312} C_VEL
LIN {X 0,Y 537.102,Z 1149.646,A -85,B 0,C 180,E1 24554.008,E2 24554.008} C_VEL
LIN {X 0,Y 537.863,Z 1142.026,A -85,B 0,C 180,E1 24551.797,E2 24551.797} C_VEL
LIN {X 0,Y 538.897,Z 1133.179,A -85,B 0,C 180,E1 24549.554,E2 24549.554} C_VEL
LIN {X 0,Y 540.187,Z 1123.369,A -85,B 0,C 180,E1 24547.357,E2 24547.357} C_VEL
LIN {X 0,Y 541.963,Z 1111.552,A -85,B 0,C 180,E1 24545.01,E2 24545.01} C_VEL
LIN {X 0,Y 544.789,Z 1094.669,A -85,B 0,C 180,E1 24542.096,E2 24542.096} C_VEL
LIN {X 0,Y 547.328,Z 1080.566,A -85,B 0,C 180,E1 24539.965,E2 24539.965} C_VEL
LIN {X 0,Y 550,Z 1066.557,A -85,B 0,C 180,E1 24538.062,E2 24538.062} C_VEL
LIN {X 0,Y 552.843,Z 1051.995,A -85,B 0,C 180,E1 24536.274,E2 24536.274} C_VEL
LIN {X 0,Y 555.164,Z 1039.961,A -85,B 0,C 180,E1 24534.935,E2 24534.935} C_VEL
LIN {X 0,Y 558.35,Z 1021.584,A -85,B 0,C 180,E1 24533.177,E2 24533.177} C_VEL
LIN {X 0,Y 561.753,Z 1001.267,A -85,B 0,C 180,E1 24531.468,E2 24531.468} C_VEL
LIN {X 0,Y 564.231,Z 985.205,A -85,B 0,C 180,E1 24530.274,E2 24530.274} C_VEL
LIN {X 0,Y 566.872,Z 966.734,A -85,B 0,C 180,E1 24529.058,E2 24529.058} C_VEL
LIN {X 0,Y 569.57,Z 946.877,A -85,B 0,C 180,E1 24527.889,E2 24527.889} C_VEL
LIN {X 0,Y 572.667,Z 921.656,A -85,B 0,C 180,E1 24526.605,E2 24526.605} C_VEL
LIN {X 0,Y 575.006,Z 899.386,A -85,B 0,C 180,E1 24525.652,E2 24525.652} C_VEL
LIN {X 0,Y 577.033,Z 878.501,A -85,B 0,C 180,E1 24524.872,E2 24524.872} C_VEL
LIN {X 0,Y 579.381,Z 851.961,A -85,B 0,C 180,E1 24524.03,E2 24524.03} C_VEL
LIN {X 0,Y 581.522,Z 822.98,A -85,B 0,C 180,E1 24523.3,E2 24523.3} C_VEL
LIN {X 0,Y 583.744,Z 787.584,A -85,B 0,C 180,E1 24522.615,E2 24522.615} C_VEL
LIN {X 0,Y 596.365,Z 577.817,A -85,B 0,C 180,E1 24518.946,E2 24518.946} C_VEL
LIN {X 0,Y 601.977,Z 473.916,A -85,B 0,C 180,E1 24517.27,E2 24517.27} C_VEL
LIN {X 0,Y 604.001,Z 425.52,A -85,B 0,C 180,E1 24516.522,E2 24516.522} C_VEL
LIN {X 0,Y 593.701,Z 415.688,A -85,B 0,C 180,E1 24514.933,E2 24514.933} C_VEL
LIN {X 0,Y 586.282,Z 408.844,A -85,B 0,C 180,E1 24513.72,E2 24513.72} C_VEL
LIN {X 0,Y 579.814,Z 403.138,A -85,B 0,C 180,E1 24512.609,E2 24512.609} C_VEL
LIN {X 0,Y 574.45,Z 398.102,A -85,B 0,C 180,E1 24511.596,E2 24511.596} C_VEL
LIN {X 0,Y 571.883,Z 393.321,A -85,B 0,C 180,E1 24509.666,E2 24509.666} C_VEL
LIN {X 0,Y 569.235,Z 388.525,A -85,B 0,C 180,E1 24507.401,E2 24507.401} C_VEL
LIN {X 0,Y 566.46,Z 383.55,A -85,B 0,C 180,E1 24504.508,E2 24504.508} C_VEL
LIN {X 0,Y 565.707,Z 382.429,A -85,B 0,C 180,E1 24503.655,E2 24503.655} C_VEL
LIN {X 0,Y 563.307,Z 377.65,A -85,B 0,C 180,E1 24499.386,E2 24499.386} C_VEL
LIN {X 0,Y 561.877,Z 376.264,A -85,B 0,C 180,E1 24494.743,E2 24494.743} C_VEL
LIN {X 0,Y 562.454,Z 376.904,A -85,B 0,C 180,E1 24490.758,E2 24490.758} C_VEL
LIN {X 0,Y 563.596,Z 378.122,A -85,B 0,C 180,E1 24488.365,E2 24488.365} C_VEL
LIN {X 0,Y 566.595,Z 383.454,A -85,B 0,C 180,E1 24483.845,E2 24483.845} C_VEL
LIN {X 0,Y 568.829,Z 387.741,A -85,B 0,C 180,E1 24481.41,E2 24481.41} C_VEL
LIN {X 0,Y 569.599,Z 389.108,A -85,B 0,C 180,E1 24480.704,E2 24480.704} C_VEL
LIN {X 0,Y 572.401,Z 394.134,A -85,B 0,C 180,E1 24478.398,E2 24478.398} C_VEL
LIN {X 0,Y 575.12,Z 399.236,A -85,B 0,C 180,E1 24476.412,E2 24476.412} C_VEL
LIN {X 0,Y 577.688,Z 404.023,A -85,B 0,C 180,E1 24474.737,E2 24474.737} C_VEL
LIN {X 0,Y 580.581,Z 409.669,A -85,B 0,C 180,E1 24472.976,E2 24472.976} C_VEL
LIN {X 0,Y 583.025,Z 414.349,A -85,B 0,C 180,E1 24471.618,E2 24471.618} C_VEL
LIN {X 0,Y 586.919,Z 421.983,A -85,B 0,C 180,E1 24469.596,E2 24469.596} C_VEL
LIN {X 0,Y 592.675,Z 433.84,A -85,B 0,C 180,E1 24466.835,E2 24466.835} C_VEL
LIN {X 0,Y 598.366,Z 446.333,A -85,B 0,C 180,E1 24464.294,E2 24464.294} C_VEL
LIN {X 0,Y 599.136,Z 448.47,A -85,B 0,C 180,E1 24463.917,E2 24463.917} C_VEL
LIN {X 0,Y 593.463,Z 483.658,A -85,B 0,C 180,E1 24460.871,E2 24460.871} C_VEL
LIN {X 0,Y 588.177,Z 518.51,A -85,B 0,C 180,E1 24457.985,E2 24457.985} C_VEL
LIN {X 0,Y 582.903,Z 556.067,A -85,B 0,C 180,E1 24454.981,E2 24454.981} C_VEL
LIN {X 0,Y 578.004,Z 597.079,A -85,B 0,C 180,E1 24451.757,E2 24451.757} C_VEL
LIN {X 0,Y 577.8,Z 615.339,A -85,B 0,C 180,E1 24450.164,E2 24450.164} C_VEL
LIN {X 0,Y 579.511,Z 631.623,A -85,B 0,C 180,E1 24448.596,E2 24448.596} C_VEL
LIN {X 0,Y 582.976,Z 646.12,A -85,B 0,C 180,E1 24447.064,E2 24447.064} C_VEL
LIN {X 0,Y 587.84,Z 658.718,A -85,B 0,C 180,E1 24445.617,E2 24445.617} C_VEL
LIN {X 0,Y 595.243,Z 671.713,A -85,B 0,C 180,E1 24443.989,E2 24443.989} C_VEL
LIN {X 0,Y 603.577,Z 682.161,A -85,B 0,C 180,E1 24442.557,E2 24442.557} C_VEL
LIN {X 0,Y 614.186,Z 692.083,A -85,B 0,C 180,E1 24441.067,E2 24441.067} C_VEL
LIN {X 0,Y 623.437,Z 698.881,A -85,B 0,C 180,E1 24439.96,E2 24439.96} C_VEL
LIN {X 0,Y 616.67,Z 708.859,A -85,B 0,C 180,E1 24439.716,E2 24439.716} C_VEL
LIN {X 0,Y 606.91,Z 722.385,A -85,B 0,C 180,E1 24439.417,E2 24439.417} C_VEL
LIN {X 0,Y 598.791,Z 735.878,A -85,B 0,C 180,E1 24439.002,E2 24439.002} C_VEL
LIN {X 0,Y 596.935,Z 739.8,A -85,B 0,C 180,E1 24438.881,E2 24438.881} C_VEL
LIN {X 0,Y 594.304,Z 755.614,A -85,B 0,C 180,E1 24438.892,E2 24438.892} C_VEL
LIN {X 0,Y 592.61,Z 772.489,A -85,B 0,C 180,E1 24438.783,E2 24438.783} C_VEL
LIN {X 0,Y 590.966,Z 814.876,A -85,B 0,C 180,E1 24438.158,E2 24438.158} C_VEL
LIN {X 0,Y 588.489,Z 847.671,A -85,B 0,C 180,E1 24437.544,E2 24437.544} C_VEL
LIN {X 0,Y 585.731,Z 877.451,A -85,B 0,C 180,E1 24436.8,E2 24436.8} C_VEL
LIN {X 0,Y 582.789,Z 905.162,A -85,B 0,C 180,E1 24435.924,E2 24435.924} C_VEL
LIN {X 0,Y 579.509,Z 931.811,A -85,B 0,C 180,E1 24434.883,E2 24434.883} C_VEL
LIN {X 0,Y 575.954,Z 956.847,A -85,B 0,C 180,E1 24433.703,E2 24433.703} C_VEL
LIN {X 0,Y 572.275,Z 980.138,A -85,B 0,C 180,E1 24432.407,E2 24432.407} C_VEL
LIN {X 0,Y 568.213,Z 1003.507,A -85,B 0,C 180,E1 24430.888,E2 24430.888} C_VEL
LIN {X 0,Y 564.937,Z 1021.1,A -85,B 0,C 180,E1 24429.579,E2 24429.579} C_VEL
LIN {X 0,Y 560.767,Z 1042.506,A -85,B 0,C 180,E1 24427.767,E2 24427.767} C_VEL
LIN {X 0,Y 557.011,Z 1061.483,A -85,B 0,C 180,E1 24425.942,E2 24425.942} C_VEL
LIN {X 0,Y 553.087,Z 1081.063,A -85,B 0,C 180,E1 24423.802,E2 24423.802} C_VEL
LIN {X 0,Y 549.559,Z 1098.858,A -85,B 0,C 180,E1 24421.599,E2 24421.599} C_VEL
LIN {X 0,Y 546.557,Z 1114.981,A -85,B 0,C 180,E1 24419.358,E2 24419.358} C_VEL
LIN {X 0,Y 543.658,Z 1131.22,A -85,B 0,C 180,E1 24416.78,E2 24416.78} C_VEL
LIN {X 0,Y 541.474,Z 1144.943,A -85,B 0,C 180,E1 24414.316,E2 24414.316} C_VEL
LIN {X 0,Y 539.519,Z 1158.47,A -85,B 0,C 180,E1 24411.509,E2 24411.509} C_VEL
LIN {X 0,Y 538.113,Z 1169.867,A -85,B 0,C 180,E1 24408.749,E2 24408.749} C_VEL
LIN {X 0,Y 537.088,Z 1179.91,A -85,B 0,C 180,E1 24405.881,E2 24405.881} C_VEL
LIN {X 0,Y 536.502,Z 1187.91,A -85,B 0,C 180,E1 24403.141,E2 24403.141} C_VEL
LIN {X 0,Y 536.143,Z 1194.477,A -85,B 0,C 180,E1 24400.312,E2 24400.312} C_VEL
LIN {X 0,Y 535.982,Z 1199.401,A -85,B 0,C 180,E1 24397.502,E2 24397.502} C_VEL
LIN {X 0,Y 535.919,Z 1202.796,A -85,B 0,C 180,E1 24394.707,E2 24394.707} C_VEL
LIN {X 0,Y 535.911,Z 1204.564,A -85,B 0,C 180,E1 24392.03,E2 24392.03} C_VEL
LIN {X 0,Y 535.899,Z 1204.88,A -85,B 0,C 180,E1 24389.25,E2 24389.25} C_VEL
LIN {X 0,Y 535.916,Z 1203.836,A -85,B 0,C 180,E1 24386.576,E2 24386.576} C_VEL
LIN {X 0,Y 535.942,Z 1201.278,A -85,B 0,C 180,E1 24383.894,E2 24383.894} C_VEL
LIN {X 0,Y 536.042,Z 1197.123,A -85,B 0,C 180,E1 24381.092,E2 24381.092} C_VEL
LIN {X 0,Y 536.275,Z 1191.66,A -85,B 0,C 180,E1 24378.382,E2 24378.382} C_VEL
LIN {X 0,Y 536.732,Z 1184.509,A -85,B 0,C 180,E1 24375.633,E2 24375.633} C_VEL
LIN {X 0,Y 537.543,Z 1175.116,A -85,B 0,C 180,E1 24372.684,E2 24372.684} C_VEL
LIN {X 0,Y 538.734,Z 1164.537,A -85,B 0,C 180,E1 24369.908,E2 24369.908} C_VEL
LIN {X 0,Y 540.313,Z 1152.718,A -85,B 0,C 180,E1 24367.245,E2 24367.245} C_VEL
LIN {X 0,Y 542.409,Z 1138.909,A -85,B 0,C 180,E1 24364.562,E2 24364.562} C_VEL
LIN {X 0,Y 545.083,Z 1122.98,A -85,B 0,C 180,E1 24361.871,E2 24361.871} C_VEL
LIN {X 0,Y 547.864,Z 1107.941,A -85,B 0,C 180,E1 24359.632,E2 24359.632} C_VEL
LIN {X 0,Y 551.366,Z 1089.551,A -85,B 0,C 180,E1 24357.218,E2 24357.218} C_VEL
LIN {X 0,Y 555.415,Z 1069.436,A -85,B 0,C 180,E1 24354.887,E2 24354.887} C_VEL
LIN {X 0,Y 559.269,Z 1050.298,A -85,B 0,C 180,E1 24352.95,E2 24352.95} C_VEL
LIN {X 0,Y 563.287,Z 1029.864,A -85,B 0,C 180,E1 24351.133,E2 24351.133} C_VEL
LIN {X 0,Y 566.982,Z 1010.795,A -85,B 0,C 180,E1 24349.627,E2 24349.627} C_VEL
LIN {X 0,Y 570.956,Z 988.379,A -85,B 0,C 180,E1 24348.098,E2 24348.098} C_VEL
LIN {X 0,Y 574.756,Z 965.12,A -85,B 0,C 180,E1 24346.73,E2 24346.73} C_VEL
LIN {X 0,Y 578.379,Z 940.219,A -85,B 0,C 180,E1 24345.49,E2 24345.49} C_VEL
LIN {X 0,Y 581.773,Z 913.715,A -85,B 0,C 180,E1 24344.388,E2 24344.388} C_VEL
LIN {X 0,Y 584.805,Z 886.502,A -85,B 0,C 180,E1 24343.464,E2 24343.464} C_VEL
LIN {X 0,Y 587.67,Z 857.065,A -85,B 0,C 180,E1 24342.67,E2 24342.67} C_VEL
LIN {X 0,Y 590.221,Z 826.171,A -85,B 0,C 180,E1 24342.037,E2 24342.037} C_VEL
LIN {X 0,Y 592.064,Z 790.181,A -85,B 0,C 180,E1 24341.462,E2 24341.462} C_VEL
LIN {X 0,Y 594.42,Z 726.683,A -85,B 0,C 180,E1 24340.572,E2 24340.572} C_VEL
LIN {X 0,Y 600.823,Z 659.715,A -85,B 0,C 180,E1 24339.444,E2 24339.444} C_VEL
LIN {X 0,Y 605.247,Z 614.722,A -85,B 0,C 180,E1 24338.699,E2 24338.699} C_VEL
LIN {X 0,Y 607.239,Z 596.992,A -85,B 0,C 180,E1 24338.433,E2 24338.433} C_VEL
LIN {X 0,Y 610.074,Z 567.332,A -85,B 0,C 180,E1 24337.933,E2 24337.933} C_VEL
LIN {X 0,Y 613.529,Z 539.192,A -85,B 0,C 180,E1 24337.545,E2 24337.545} C_VEL
LIN {X 0,Y 615.973,Z 512.739,A -85,B 0,C 180,E1 24337.09,E2 24337.09} C_VEL
LIN {X 0,Y 620.663,Z 476.513,A -85,B 0,C 180,E1 24336.62,E2 24336.62} C_VEL
LIN {X 0,Y 622.607,Z 453.394,A -85,B 0,C 180,E1 24336.2,E2 24336.2} C_VEL
LIN {X 0,Y 615.066,Z 442.583,A -85,B 0,C 180,E1 24334.987,E2 24334.987} C_VEL
LIN {X 0,Y 602.567,Z 423.116,A -85,B 0,C 180,E1 24332.777,E2 24332.777} C_VEL
LIN {X 0,Y 590.763,Z 405.799,A -85,B 0,C 180,E1 24330.515,E2 24330.515} C_VEL
LIN {X 0,Y 579.608,Z 390.336,A -85,B 0,C 180,E1 24328.181,E2 24328.181} C_VEL
LIN {X 0,Y 570.777,Z 378.851,A -85,B 0,C 180,E1 24326.169,E2 24326.169} C_VEL
LIN {X 0,Y 566.679,Z 373.503,A -85,B 0,C 180,E1 24325.166,E2 24325.166} C_VEL
LIN {X 0,Y 563.105,Z 368.703,A -85,B 0,C 180,E1 24324.244,E2 24324.244} C_VEL
LIN {X 0,Y 559.287,Z 364.312,A -85,B 0,C 180,E1 24323.245,E2 24323.245} C_VEL
LIN {X 0,Y 558.017,Z 362.447,A -85,B 0,C 180,E1 24322.882,E2 24322.882} C_VEL
LIN {X 0,Y 554.688,Z 358.932,A -85,B 0,C 180,E1 24321.965,E2 24321.965} C_VEL
LIN {X 0,Y 553.111,Z 356.411,A -85,B 0,C 180,E1 24321.474,E2 24321.474} C_VEL
LIN {X 0,Y 549.924,Z 353.341,A -85,B 0,C 180,E1 24320.544,E2 24320.544} C_VEL
LIN {X 0,Y 548.195,Z 350.231,A -85,B 0,C 180,E1 24319.943,E2 24319.943} C_VEL
LIN {X 0,Y 544.972,Z 347.709,A -85,B 0,C 180,E1 24318.951,E2 24318.951} C_VEL
LIN {X 0,Y 543.182,Z 344.38,A -85,B 0,C 180,E1 24318.264,E2 24318.264} C_VEL
LIN {X 0,Y 542.855,Z 343.786,A -85,B 0,C 180,E1 24318.137,E2 24318.137} C_VEL
LIN {X 0,Y 539.692,Z 341.691,A -85,B 0,C 180,E1 24317.077,E2 24317.077} C_VEL
LIN {X 0,Y 537.96,Z 338.793,A -85,B 0,C 180,E1 24316.355,E2 24316.355} C_VEL
LIN {X 0,Y 537.84,Z 338.395,A -85,B 0,C 180,E1 24316.262,E2 24316.262} C_VEL
LIN {X 0,Y 545.247,Z 358.462,A -85,B 0,C 180,E1 24315.178,E2 24315.178} C_VEL
LIN {X 0,Y 545.696,Z 361.534,A -85,B 0,C 180,E1 24315.048,E2 24315.048} C_VEL
LIN {X 0,Y 545.263,Z 442.105,A -85,B 0,C 180,E1 24312.121,E2 24312.121} C_VEL
LIN {X 0,Y 545.327,Z 522.138,A -85,B 0,C 180,E1 24309.073,E2 24309.073} C_VEL
LIN {X 0,Y 544.943,Z 598.444,A -85,B 0,C 180,E1 24306.083,E2 24306.083} C_VEL
LIN {X 0,Y 544.187,Z 675.062,A -85,B 0,C 180,E1 24303.002,E2 24303.002} C_VEL
LIN {X 0,Y 543.087,Z 753.187,A -85,B 0,C 180,E1 24299.789,E2 24299.789} C_VEL
LIN {X 0,Y 541.88,Z 832.759,A -85,B 0,C 180,E1 24296.456,E2 24296.456} C_VEL
LIN {X 0,Y 541.242,Z 853.144,A -85,B 0,C 180,E1 24295.603,E2 24295.603} C_VEL
LIN {X 0,Y 540.559,Z 862.859,A -85,B 0,C 180,E1 24295.237,E2 24295.237} C_VEL
LIN {X 0,Y 539.69,Z 975.636,A -85,B 0,C 180,E1 24293.604,E2 24293.604} C_VEL
LIN {X 0,Y 539.741,Z 988.613,A -85,B 0,C 180,E1 24293.279,E2 24293.279} C_VEL
LIN {X 0,Y 539.706,Z 999.922,A -85,B 0,C 180,E1 24292.87,E2 24292.87} C_VEL
LIN {X 0,Y 539.568,Z 1012.157,A -85,B 0,C 180,E1 24292.279,E2 24292.279} C_VEL
LIN {X 0,Y 539.305,Z 1025.458,A -85,B 0,C 180,E1 24291.416,E2 24291.416} C_VEL
LIN {X 0,Y 539.04,Z 1035.218,A -85,B 0,C 180,E1 24290.605,E2 24290.605} C_VEL
LIN {X 0,Y 538.758,Z 1043.771,A -85,B 0,C 180,E1 24289.737,E2 24289.737} C_VEL
LIN {X 0,Y 538.498,Z 1050.869,A -85,B 0,C 180,E1 24288.866,E2 24288.866} C_VEL
LIN {X 0,Y 538.236,Z 1057.478,A -85,B 0,C 180,E1 24287.882,E2 24287.882} C_VEL
LIN {X 0,Y 537.985,Z 1063.422,A -85,B 0,C 180,E1 24286.785,E2 24286.785} C_VEL
LIN {X 0,Y 537.737,Z 1069.349,A -85,B 0,C 180,E1 24285.352,E2 24285.352} C_VEL
LIN {X 0,Y 537.546,Z 1073.244,A -85,B 0,C 180,E1 24283.909,E2 24283.909} C_VEL
LIN {X 0,Y 537.445,Z 1075.328,A -85,B 0,C 180,E1 24282.634,E2 24282.634} C_VEL
LIN {X 0,Y 537.387,Z 1076.148,A -85,B 0,C 180,E1 24281.448,E2 24281.448} C_VEL
LIN {X 0,Y 537.371,Z 1075.867,A -85,B 0,C 180,E1 24280.205,E2 24280.205} C_VEL
LIN {X 0,Y 537.405,Z 1074.074,A -85,B 0,C 180,E1 24278.727,E2 24278.727} C_VEL
LIN {X 0,Y 537.516,Z 1070.434,A -85,B 0,C 180,E1 24277.237,E2 24277.237} C_VEL
LIN {X 0,Y 537.662,Z 1065.762,A -85,B 0,C 180,E1 24275.94,E2 24275.94} C_VEL
LIN {X 0,Y 537.858,Z 1060.39,A -85,B 0,C 180,E1 24274.804,E2 24274.804} C_VEL
LIN {X 0,Y 538.141,Z 1053.104,A -85,B 0,C 180,E1 24273.584,E2 24273.584} C_VEL
LIN {X 0,Y 538.513,Z 1043.087,A -85,B 0,C 180,E1 24272.288,E2 24272.288} C_VEL
LIN {X 0,Y 538.817,Z 1034.223,A -85,B 0,C 180,E1 24271.373,E2 24271.373} C_VEL
LIN {X 0,Y 539.103,Z 1024.657,A -85,B 0,C 180,E1 24270.56,E2 24270.56} C_VEL
LIN {X 0,Y 539.365,Z 1014.315,A -85,B 0,C 180,E1 24269.842,E2 24269.842} C_VEL
LIN {X 0,Y 539.643,Z 1001.198,A -85,B 0,C 180,E1 24269.12,E2 24269.12} C_VEL
LIN {X 0,Y 539.777,Z 986.629,A -85,B 0,C 180,E1 24268.554,E2 24268.554} C_VEL
LIN {X 0,Y 539.799,Z 974.2,A -85,B 0,C 180,E1 24268.223,E2 24268.223} C_VEL
LIN {X 0,Y 539.769,Z 952.012,A -85,B 0,C 180,E1 24267.874,E2 24267.874} C_VEL
LIN {X 0,Y 540.808,Z 855.419,A -85,B 0,C 180,E1 24266.497,E2 24266.497} C_VEL
LIN {X 0,Y 541.566,Z 840.438,A -85,B 0,C 180,E1 24265.856,E2 24265.856} C_VEL
LIN {X 0,Y 543.209,Z 762.94,A -85,B 0,C 180,E1 24262.431,E2 24262.431} C_VEL
LIN {X 0,Y 544.119,Z 764.234,A -85,B 0,C 180,E1 24262.27,E2 24262.27} C_VEL
LIN {X 0,Y 545.706,Z 764.132,A -85,B 0,C 180,E1 24262.067,E2 24262.067} C_VEL
LIN {X 0,Y 548.389,Z 761.711,A -85,B 0,C 180,E1 24261.8,E2 24261.8} C_VEL
LIN {X 0,Y 552.069,Z 755.962,A -85,B 0,C 180,E1 24261.519,E2 24261.519} C_VEL
LIN {X 0,Y 552.818,Z 754.961,A -85,B 0,C 180,E1 24261.457,E2 24261.457} C_VEL
LIN {X 0,Y 556.124,Z 753.286,A -85,B 0,C 180,E1 24261.102,E2 24261.102} C_VEL
LIN {X 0,Y 559.954,Z 749.311,A -85,B 0,C 180,E1 24260.76,E2 24260.76} C_VEL
LIN {X 0,Y 563.06,Z 744.776,A -85,B 0,C 180,E1 24260.525,E2 24260.525} C_VEL
LIN {X 0,Y 567.448,Z 741.723,A -85,B 0,C 180,E1 24260.104,E2 24260.104} C_VEL
LIN {X 0,Y 572.004,Z 736.51,A -85,B 0,C 180,E1 24259.733,E2 24259.733} C_VEL
LIN {X 0,Y 573.853,Z 734.084,A -85,B 0,C 180,E1 24259.595,E2 24259.595} C_VEL
LIN {X 0,Y 579.079,Z 729.919,A -85,B 0,C 180,E1 24259.139,E2 24259.139} C_VEL
LIN {X 0,Y 584.84,Z 723.306,A -85,B 0,C 180,E1 24258.705,E2 24258.705} C_VEL
LIN {X 0,Y 587.552,Z 721.442,A -85,B 0,C 180,E1 24258.476,E2 24258.476} C_VEL
LIN {X 0,Y 586.009,Z 747.445,A -85,B 0,C 180,E1 24258.01,E2 24258.01} C_VEL
LIN {X 0,Y 584.859,Z 755.09,A -85,B 0,C 180,E1 24257.941,E2 24257.941} C_VEL
LIN {X 0,Y 579.111,Z 775.539,A -85,B 0,C 180,E1 24257.997,E2 24257.997} C_VEL
LIN {X 0,Y 578.146,Z 782.095,A -85,B 0,C 180,E1 24257.929,E2 24257.929} C_VEL
LIN {X 0,Y 575.528,Z 821.158,A -85,B 0,C 180,E1 24257.166,E2 24257.166} C_VEL
LIN {X 0,Y 573.317,Z 846.681,A -85,B 0,C 180,E1 24256.498,E2 24256.498} C_VEL
LIN {X 0,Y 570.784,Z 873.028,A -85,B 0,C 180,E1 24255.656,E2 24255.656} C_VEL
LIN {X 0,Y 567.721,Z 902.253,A -85,B 0,C 180,E1 24254.542,E2 24254.542} C_VEL
LIN {X 0,Y 564.598,Z 929.912,A -85,B 0,C 180,E1 24253.291,E2 24253.291} C_VEL
LIN {X 0,Y 561.677,Z 952.967,A -85,B 0,C 180,E1 24252.069,E2 24252.069} C_VEL
LIN {X 0,Y 559.095,Z 971.322,A -85,B 0,C 180,E1 24250.955,E2 24250.955} C_VEL
LIN {X 0,Y 555.488,Z 995.289,A -85,B 0,C 180,E1 24249.284,E2 24249.284} C_VEL
LIN {X 0,Y 552.435,Z 1014.094,A -85,B 0,C 180,E1 24247.784,E2 24247.784} C_VEL
LIN {X 0,Y 549.312,Z 1032.106,A -85,B 0,C 180,E1 24246.141,E2 24246.141} C_VEL
LIN {X 0,Y 545.93,Z 1050.672,A -85,B 0,C 180,E1 24244.215,E2 24244.215} C_VEL
LIN {X 0,Y 543.676,Z 1062.753,A -85,B 0,C 180,E1 24242.808,E2 24242.808} C_VEL
LIN {X 0,Y 540.682,Z 1077.584,A -85,B 0,C 180,E1 24240.815,E2 24240.815} C_VEL
LIN {X 0,Y 538.16,Z 1090.522,A -85,B 0,C 180,E1 24238.887,E2 24238.887} C_VEL
LIN {X 0,Y 535.87,Z 1102.885,A -85,B 0,C 180,E1 24236.844,E2 24236.844} C_VEL
LIN {X 0,Y 533.914,Z 1114.374,A -85,B 0,C 180,E1 24234.73,E2 24234.73} C_VEL
LIN {X 0,Y 532.317,Z 1124.517,A -85,B 0,C 180,E1 24232.649,E2 24232.649} C_VEL
LIN {X 0,Y 531.024,Z 1133.862,A -85,B 0,C 180,E1 24230.502,E2 24230.502} C_VEL
LIN {X 0,Y 529.951,Z 1142.526,A -85,B 0,C 180,E1 24228.253,E2 24228.253} C_VEL
LIN {X 0,Y 529.12,Z 1150.512,A -85,B 0,C 180,E1 24225.872,E2 24225.872} C_VEL
LIN {X 0,Y 528.556,Z 1157.725,A -85,B 0,C 180,E1 24223.345,E2 24223.345} C_VEL
LIN {X 0,Y 528.15,Z 1164.832,A -85,B 0,C 180,E1 24220.252,E2 24220.252} C_VEL
LIN {X 0,Y 527.98,Z 1169.466,A -85,B 0,C 180,E1 24217.51,E2 24217.51} C_VEL
LIN {X 0,Y 527.925,Z 1172.481,A -85,B 0,C 180,E1 24214.999,E2 24214.999} C_VEL
LIN {X 0,Y 527.907,Z 1174.241,A -85,B 0,C 180,E1 24212.607,E2 24212.607} C_VEL
LIN {X 0,Y 527.901,Z 1174.905,A -85,B 0,C 180,E1 24210.218,E2 24210.218} C_VEL
LIN {X 0,Y 527.911,Z 1174.477,A -85,B 0,C 180,E1 24207.83,E2 24207.83} C_VEL
LIN {X 0,Y 527.918,Z 1173.052,A -85,B 0,C 180,E1 24205.548,E2 24205.548} C_VEL
LIN {X 0,Y 527.954,Z 1170.618,A -85,B 0,C 180,E1 24203.258,E2 24203.258} C_VEL
LIN {X 0,Y 528.055,Z 1166.967,A -85,B 0,C 180,E1 24200.849,E2 24200.849} C_VEL
LIN {X 0,Y 528.249,Z 1162.413,A -85,B 0,C 180,E1 24198.538,E2 24198.538} C_VEL
LIN {X 0,Y 528.615,Z 1156.774,A -85,B 0,C 180,E1 24196.213,E2 24196.213} C_VEL
LIN {X 0,Y 529.164,Z 1149.996,A -85,B 0,C 180,E1 24193.875,E2 24193.875} C_VEL
LIN {X 0,Y 529.963,Z 1142.417,A -85,B 0,C 180,E1 24191.627,E2 24191.627} C_VEL
LIN {X 0,Y 531.051,Z 1133.646,A -85,B 0,C 180,E1 24189.355,E2 24189.355} C_VEL
LIN {X 0,Y 532.335,Z 1124.409,A -85,B 0,C 180,E1 24187.238,E2 24187.238} C_VEL
LIN {X 0,Y 533.893,Z 1114.466,A -85,B 0,C 180,E1 24185.198,E2 24185.198} C_VEL
LIN {X 0,Y 535.8,Z 1103.251,A -85,B 0,C 180,E1 24183.13,E2 24183.13} C_VEL
LIN {X 0,Y 538.097,Z 1090.826,A -85,B 0,C 180,E1 24181.07,E2 24181.07} C_VEL
LIN {X 0,Y 540.722,Z 1077.389,A -85,B 0,C 180,E1 24179.067,E2 24179.067} C_VEL
LIN {X 0,Y 543.891,Z 1061.672,A -85,B 0,C 180,E1 24176.963,E2 24176.963} C_VEL
LIN {X 0,Y 547.521,Z 1041.979,A -85,B 0,C 180,E1 24174.757,E2 24174.757} C_VEL
LIN {X 0,Y 551.387,Z 1020.392,A -85,B 0,C 180,E1 24172.671,E2 24172.671} C_VEL
LIN {X 0,Y 554.456,Z 1001.819,A -85,B 0,C 180,E1 24171.131,E2 24171.131} C_VEL
LIN {X 0,Y 557.196,Z 984.161,A -85,B 0,C 180,E1 24169.828,E2 24169.828} C_VEL
LIN {X 0,Y 559.963,Z 965.477,A -85,B 0,C 180,E1 24168.588,E2 24168.588} C_VEL
LIN {X 0,Y 562.867,Z 944.071,A -85,B 0,C 180,E1 24167.345,E2 24167.345} C_VEL
LIN {X 0,Y 565.77,Z 919.778,A -85,B 0,C 180,E1 24166.143,E2 24166.143} C_VEL
LIN {X 0,Y 568.114,Z 898.469,A -85,B 0,C 180,E1 24165.218,E2 24165.218} C_VEL
LIN {X 0,Y 571.194,Z 868.447,A -85,B 0,C 180,E1 24164.1,E2 24164.1} C_VEL
LIN {X 0,Y 573.515,Z 844.452,A -85,B 0,C 180,E1 24163.348,E2 24163.348} C_VEL
LIN {X 0,Y 575.86,Z 816.581,A -85,B 0,C 180,E1 24162.642,E2 24162.642} C_VEL
LIN {X 0,Y 581.116,Z 735.117,A -85,B 0,C 180,E1 24161.115,E2 24161.115} C_VEL
LIN {X 0,Y 590.81,Z 586.822,A -85,B 0,C 180,E1 24158.491,E2 24158.491} C_VEL
LIN {X 0,Y 596.572,Z 486.507,A -85,B 0,C 180,E1 24156.849,E2 24156.849} C_VEL
LIN {X 0,Y 599.083,Z 430.582,A -85,B 0,C 180,E1 24155.98,E2 24155.98} C_VEL
LIN {X 0,Y 586.4,Z 418.403,A -85,B 0,C 180,E1 24153.948,E2 24153.948} C_VEL
LIN {X 0,Y 577.441,Z 410.501,A -85,B 0,C 180,E1 24152.407,E2 24152.407} C_VEL
LIN {X 0,Y 570.974,Z 404.826,A -85,B 0,C 180,E1 24151.222,E2 24151.222} C_VEL
LIN {X 0,Y 568.781,Z 403.025,A -85,B 0,C 180,E1 24150.768,E2 24150.768} C_VEL
LIN {X 0,Y 566.874,Z 399.131,A -85,B 0,C 180,E1 24149.182,E2 24149.182} C_VEL
LIN {X 0,Y 564.315,Z 394.374,A -85,B 0,C 180,E1 24146.861,E2 24146.861} C_VEL
LIN {X 0,Y 562.099,Z 390.128,A -85,B 0,C 180,E1 24144.374,E2 24144.374} C_VEL
LIN {X 0,Y 559.06,Z 384.424,A -85,B 0,C 180,E1 24139.322,E2 24139.322} C_VEL
LIN {X 0,Y 557.686,Z 383.079,A -85,B 0,C 180,E1 24134.75,E2 24134.75} C_VEL
LIN {X 0,Y 558.269,Z 383.727,A -85,B 0,C 180,E1 24130.735,E2 24130.735} C_VEL
LIN {X 0,Y 559.385,Z 385.011,A -85,B 0,C 180,E1 24128.325,E2 24128.325} C_VEL
LIN {X 0,Y 562.302,Z 390.257,A -85,B 0,C 180,E1 24123.875,E2 24123.875} C_VEL
LIN {X 0,Y 564.555,Z 394.508,A -85,B 0,C 180,E1 24121.421,E2 24121.421} C_VEL
LIN {X 0,Y 565.362,Z 396.194,A -85,B 0,C 180,E1 24120.608,E2 24120.608} C_VEL
LIN {X 0,Y 567.949,Z 400.741,A -85,B 0,C 180,E1 24118.487,E2 24118.487} C_VEL
LIN {X 0,Y 570.634,Z 405.857,A -85,B 0,C 180,E1 24116.484,E2 24116.484} C_VEL
LIN {X 0,Y 573.172,Z 410.664,A -85,B 0,C 180,E1 24114.795,E2 24114.795} C_VEL
LIN {X 0,Y 577.511,Z 418.808,A -85,B 0,C 180,E1 24112.239,E2 24112.239} C_VEL
LIN {X 0,Y 582.313,Z 428.72,A -85,B 0,C 180,E1 24109.613,E2 24109.613} C_VEL
LIN {X 0,Y 587.63,Z 439.752,A -85,B 0,C 180,E1 24107.02,E2 24107.02} C_VEL
LIN {X 0,Y 593.242,Z 452.245,A -85,B 0,C 180,E1 24104.455,E2 24104.455} C_VEL
LIN {X 0,Y 593.616,Z 453.317,A -85,B 0,C 180,E1 24104.265,E2 24104.265} C_VEL
LIN {X 0,Y 587.785,Z 487.991,A -85,B 0,C 180,E1 24101.246,E2 24101.246} C_VEL
LIN {X 0,Y 582.265,Z 522.921,A -85,B 0,C 180,E1 24098.333,E2 24098.333} C_VEL
LIN {X 0,Y 576.726,Z 560.687,A -85,B 0,C 180,E1 24095.291,E2 24095.291} C_VEL
LIN {X 0,Y 571.822,Z 600.036,A -85,B 0,C 180,E1 24092.168,E2 24092.168} C_VEL
LIN {X 0,Y 571.485,Z 618.398,A -85,B 0,C 180,E1 24090.551,E2 24090.551} C_VEL
LIN {X 0,Y 573.07,Z 634.949,A -85,B 0,C 180,E1 24088.944,E2 24088.944} C_VEL
LIN {X 0,Y 576.472,Z 649.863,A -85,B 0,C 180,E1 24087.355,E2 24087.355} C_VEL
LIN {X 0,Y 581.596,Z 663.428,A -85,B 0,C 180,E1 24085.782,E2 24085.782} C_VEL
LIN {X 0,Y 588.892,Z 676.41,A -85,B 0,C 180,E1 24084.142,E2 24084.142} C_VEL
LIN {X 0,Y 597.137,Z 686.963,A -85,B 0,C 180,E1 24082.687,E2 24082.687} C_VEL
LIN {X 0,Y 608.227,Z 697.515,A -85,B 0,C 180,E1 24081.098,E2 24081.098} C_VEL
LIN {X 0,Y 614.359,Z 702.249,A -85,B 0,C 180,E1 24080.335,E2 24080.335} C_VEL
LIN {X 0,Y 609.738,Z 708.668,A -85,B 0,C 180,E1 24080.197,E2 24080.197} C_VEL
LIN {X 0,Y 600.132,Z 722.304,A -85,B 0,C 180,E1 24079.882,E2 24079.882} C_VEL
LIN {X 0,Y 592.268,Z 735.862,A -85,B 0,C 180,E1 24079.468,E2 24079.468} C_VEL
LIN {X 0,Y 589.077,Z 755.435,A -85,B 0,C 180,E1 24079.478,E2 24079.478} C_VEL
LIN {X 0,Y 587.344,Z 772.689,A -85,B 0,C 180,E1 24079.368,E2 24079.368} C_VEL
LIN {X 0,Y 585.641,Z 813.256,A -85,B 0,C 180,E1 24078.761,E2 24078.761} C_VEL
LIN {X 0,Y 582.961,Z 846.684,A -85,B 0,C 180,E1 24078.127,E2 24078.127} C_VEL
LIN {X 0,Y 580.043,Z 876.773,A -85,B 0,C 180,E1 24077.375,E2 24077.375} C_VEL
LIN {X 0,Y 576.98,Z 904.915,A -85,B 0,C 180,E1 24076.487,E2 24076.487} C_VEL
LIN {X 0,Y 573.73,Z 931.57,A -85,B 0,C 180,E1 24075.461,E2 24075.461} C_VEL
LIN {X 0,Y 570.223,Z 956.616,A -85,B 0,C 180,E1 24074.298,E2 24074.298} C_VEL
LIN {X 0,Y 566.314,Z 980.699,A -85,B 0,C 180,E1 24072.96,E2 24072.96} C_VEL
LIN {X 0,Y 562.366,Z 1002.621,A -85,B 0,C 180,E1 24071.536,E2 24071.536} C_VEL
LIN {X 0,Y 558.14,Z 1024.557,A -85,B 0,C 180,E1 24069.89,E2 24069.89} C_VEL
LIN {X 0,Y 554.353,Z 1042.773,A -85,B 0,C 180,E1 24068.315,E2 24068.315} C_VEL
LIN {X 0,Y 549.861,Z 1063.941,A -85,B 0,C 180,E1 24066.225,E2 24066.225} C_VEL
LIN {X 0,Y 545.371,Z 1084.96,A -85,B 0,C 180,E1 24063.846,E2 24063.846} C_VEL
LIN {X 0,Y 541.119,Z 1105.619,A -85,B 0,C 180,E1 24061.155,E2 24061.155} C_VEL
LIN {X 0,Y 537.828,Z 1122.278,A -85,B 0,C 180,E1 24058.661,E2 24058.661} C_VEL
LIN {X 0,Y 535.081,Z 1137.709,A -85,B 0,C 180,E1 24056.047,E2 24056.047} C_VEL
LIN {X 0,Y 532.709,Z 1152.211,A -85,B 0,C 180,E1 24053.212,E2 24053.212} C_VEL
LIN {X 0,Y 531,Z 1164.118,A -85,B 0,C 180,E1 24050.5,E2 24050.5} C_VEL
LIN {X 0,Y 529.711,Z 1174.737,A -85,B 0,C 180,E1 24047.691,E2 24047.691} C_VEL
LIN {X 0,Y 528.848,Z 1183.956,A -85,B 0,C 180,E1 24044.786,E2 24044.786} C_VEL
LIN {X 0,Y 528.333,Z 1191.146,A -85,B 0,C 180,E1 24042.014,E2 24042.014} C_VEL
LIN {X 0,Y 528.065,Z 1196.734,A -85,B 0,C 180,E1 24039.26,E2 24039.26} C_VEL
LIN {X 0,Y 527.955,Z 1200.908,A -85,B 0,C 180,E1 24036.523,E2 24036.523} C_VEL
LIN {X 0,Y 527.913,Z 1203.587,A -85,B 0,C 180,E1 24033.8,E2 24033.8} C_VEL
LIN {X 0,Y 527.913,Z 1204.828,A -85,B 0,C 180,E1 24031.084,E2 24031.084} C_VEL
LIN {X 0,Y 527.91,Z 1204.747,A -85,B 0,C 180,E1 24028.479,E2 24028.479} C_VEL
LIN {X 0,Y 527.918,Z 1203.233,A -85,B 0,C 180,E1 24025.763,E2 24025.763} C_VEL
LIN {X 0,Y 527.961,Z 1200.351,A -85,B 0,C 180,E1 24023.037,E2 24023.037} C_VEL
LIN {X 0,Y 528.099,Z 1195.947,A -85,B 0,C 180,E1 24020.298,E2 24020.298} C_VEL
LIN {X 0,Y 528.403,Z 1189.791,A -85,B 0,C 180,E1 24017.43,E2 24017.43} C_VEL
LIN {X 0,Y 528.988,Z 1182.329,A -85,B 0,C 180,E1 24014.654,E2 24014.654} C_VEL
LIN {X 0,Y 529.947,Z 1172.792,A -85,B 0,C 180,E1 24011.746,E2 24011.746} C_VEL
LIN {X 0,Y 531.264,Z 1162.002,A -85,B 0,C 180,E1 24008.991,E2 24008.991} C_VEL
LIN {X 0,Y 533.205,Z 1148.86,A -85,B 0,C 180,E1 24006.105,E2 24006.105} C_VEL
LIN {X 0,Y 535.605,Z 1134.496,A -85,B 0,C 180,E1 24003.381,E2 24003.381} C_VEL
LIN {X 0,Y 538.258,Z 1120.108,A -85,B 0,C 180,E1 24000.997,E2 24000.997} C_VEL
LIN {X 0,Y 541.742,Z 1102.223,A -85,B 0,C 180,E1 23998.386,E2 23998.386} C_VEL
LIN {X 0,Y 546.036,Z 1081.999,A -85,B 0,C 180,E1 23995.793,E2 23995.793} C_VEL
LIN {X 0,Y 549.975,Z 1063.376,A -85,B 0,C 180,E1 23993.716,E2 23993.716} C_VEL
LIN {X 0,Y 554.59,Z 1042.018,A -85,B 0,C 180,E1 23991.602,E2 23991.602} C_VEL
LIN {X 0,Y 558.686,Z 1021.725,A -85,B 0,C 180,E1 23989.886,E2 23989.886} C_VEL
LIN {X 0,Y 563.475,Z 997.081,A -85,B 0,C 180,E1 23988.078,E2 23988.078} C_VEL
LIN {X 0,Y 567.452,Z 974.261,A -85,B 0,C 180,E1 23986.659,E2 23986.659} C_VEL
LIN {X 0,Y 571.122,Z 950.637,A -85,B 0,C 180,E1 23985.408,E2 23985.408} C_VEL
LIN {X 0,Y 574.506,Z 925.422,A -85,B 0,C 180,E1 23984.284,E2 23984.284} C_VEL
LIN {X 0,Y 577.843,Z 897.374,A -85,B 0,C 180,E1 23983.254,E2 23983.254} C_VEL
LIN {X 0,Y 580.994,Z 867.66,A -85,B 0,C 180,E1 23982.375,E2 23982.375} C_VEL
LIN {X 0,Y 583.828,Z 836.978,A -85,B 0,C 180,E1 23981.672,E2 23981.672} C_VEL
LIN {X 0,Y 586.3,Z 800.987,A -85,B 0,C 180,E1 23981.04,E2 23981.04} C_VEL
LIN {X 0,Y 589.385,Z 722.578,A -85,B 0,C 180,E1 23979.926,E2 23979.926} C_VEL
LIN {X 0,Y 595.571,Z 659.484,A -85,B 0,C 180,E1 23978.864,E2 23978.864} C_VEL
LIN {X 0,Y 599.936,Z 615.663,A -85,B 0,C 180,E1 23978.134,E2 23978.134} C_VEL
LIN {X 0,Y 601.996,Z 597.6,A -85,B 0,C 180,E1 23977.863,E2 23977.863} C_VEL
LIN {X 0,Y 604.936,Z 567.5,A -85,B 0,C 180,E1 23977.355,E2 23977.355} C_VEL
LIN {X 0,Y 608.385,Z 539.7,A -85,B 0,C 180,E1 23976.971,E2 23976.971} C_VEL
LIN {X 0,Y 610.951,Z 512.681,A -85,B 0,C 180,E1 23976.507,E2 23976.507} C_VEL
LIN {X 0,Y 615.612,Z 477.021,A -85,B 0,C 180,E1 23976.044,E2 23976.044} C_VEL
LIN {X 0,Y 617.168,Z 457.728,A -85,B 0,C 180,E1 23975.679,E2 23975.679} C_VEL
LIN {X 0,Y 598.859,Z 429.413,A -85,B 0,C 180,E1 23972.466,E2 23972.466} C_VEL
LIN {X 0,Y 587.398,Z 412.441,A -85,B 0,C 180,E1 23970.228,E2 23970.228} C_VEL
LIN {X 0,Y 576.464,Z 397.141,A -85,B 0,C 180,E1 23967.897,E2 23967.897} C_VEL
LIN {X 0,Y 567.733,Z 385.675,A -85,B 0,C 180,E1 23965.871,E2 23965.871} C_VEL
LIN {X 0,Y 563.68,Z 380.369,A -85,B 0,C 180,E1 23964.86,E2 23964.86} C_VEL
LIN {X 0,Y 559.491,Z 374.982,A -85,B 0,C 180,E1 23963.766,E2 23963.766} C_VEL
LIN {X 0,Y 555.999,Z 370.403,A -85,B 0,C 180,E1 23962.802,E2 23962.802} C_VEL
LIN {X 0,Y 551.874,Z 365.729,A -85,B 0,C 180,E1 23961.636,E2 23961.636} C_VEL
LIN {X 0,Y 550.62,Z 363.775,A -85,B 0,C 180,E1 23961.24,E2 23961.24} C_VEL
LIN {X 0,Y 547.336,Z 360.39,A -85,B 0,C 180,E1 23960.254,E2 23960.254} C_VEL
LIN {X 0,Y 545.751,Z 357.674,A -85,B 0,C 180,E1 23959.701,E2 23959.701} C_VEL
LIN {X 0,Y 542.455,Z 354.794,A -85,B 0,C 180,E1 23958.651,E2 23958.651} C_VEL
LIN {X 0,Y 540.47,Z 351.315,A -85,B 0,C 180,E1 23957.885,E2 23957.885} C_VEL
LIN {X 0,Y 537.259,Z 348.834,A -85,B 0,C 180,E1 23956.766,E2 23956.766} C_VEL
LIN {X 0,Y 536.692,Z 348.414,A -85,B 0,C 180,E1 23956.562,E2 23956.562} C_VEL
LIN {X 0,Y 535.216,Z 350.43,A -85,B 0,C 180,E1 23956.218,E2 23956.218} C_VEL
LIN {X 0,Y 534.52,Z 350.996,A -85,B 0,C 180,E1 23955.979,E2 23955.979} C_VEL
LIN {X 0,Y 538.371,Z 362.724,A -85,B 0,C 180,E1 23955.365,E2 23955.365} C_VEL
LIN {X 0,Y 537.839,Z 450.32,A -85,B 0,C 180,E1 23952.153,E2 23952.153} C_VEL
LIN {X 0,Y 537.84,Z 530.532,A -85,B 0,C 180,E1 23949.065,E2 23949.065} C_VEL
LIN {X 0,Y 537.377,Z 600.387,A -85,B 0,C 180,E1 23946.303,E2 23946.303} C_VEL
LIN {X 0,Y 536.751,Z 659.824,A -85,B 0,C 180,E1 23943.899,E2 23943.899} C_VEL
LIN {X 0,Y 535.68,Z 739.249,A -85,B 0,C 180,E1 23940.642,E2 23940.642} C_VEL
LIN {X 0,Y 534.372,Z 822.153,A -85,B 0,C 180,E1 23937.158,E2 23937.158} C_VEL
LIN {X 0,Y 533.621,Z 852.644,A -85,B 0,C 180,E1 23935.871,E2 23935.871} C_VEL
LIN {X 0,Y 532.794,Z 864.112,A -85,B 0,C 180,E1 23935.432,E2 23935.432} C_VEL
LIN {X 0,Y 531.878,Z 976.164,A -85,B 0,C 180,E1 23933.781,E2 23933.781} C_VEL
LIN {X 0,Y 531.933,Z 989.714,A -85,B 0,C 180,E1 23933.439,E2 23933.439} C_VEL
LIN {X 0,Y 531.894,Z 1001.279,A -85,B 0,C 180,E1 23933.014,E2 23933.014} C_VEL
LIN {X 0,Y 531.755,Z 1013.077,A -85,B 0,C 180,E1 23932.436,E2 23932.436} C_VEL
LIN {X 0,Y 531.484,Z 1026.476,A -85,B 0,C 180,E1 23931.562,E2 23931.562} C_VEL
LIN {X 0,Y 531.184,Z 1036.847,A -85,B 0,C 180,E1 23930.684,E2 23930.684} C_VEL
LIN {X 0,Y 530.892,Z 1045.332,A -85,B 0,C 180,E1 23929.802,E2 23929.802} C_VEL
LIN {X 0,Y 530.589,Z 1053.181,A -85,B 0,C 180,E1 23928.808,E2 23928.808} C_VEL
LIN {X 0,Y 530.246,Z 1061.545,A -85,B 0,C 180,E1 23927.475,E2 23927.475} C_VEL
LIN {X 0,Y 529.95,Z 1067.721,A -85,B 0,C 180,E1 23926.136,E2 23926.136} C_VEL
LIN {X 0,Y 529.754,Z 1071.961,A -85,B 0,C 180,E1 23924.902,E2 23924.902} C_VEL
LIN {X 0,Y 529.605,Z 1074.934,A -85,B 0,C 180,E1 23923.661,E2 23923.661} C_VEL
LIN {X 0,Y 529.508,Z 1076.833,A -85,B 0,C 180,E1 23922.301,E2 23922.301} C_VEL
LIN {X 0,Y 529.45,Z 1077.208,A -85,B 0,C 180,E1 23920.586,E2 23920.586} C_VEL
LIN {X 0,Y 529.463,Z 1075.904,A -85,B 0,C 180,E1 23919.198,E2 23919.198} C_VEL
LIN {X 0,Y 529.525,Z 1073.478,A -85,B 0,C 180,E1 23917.928,E2 23917.928} C_VEL
LIN {X 0,Y 529.666,Z 1069.375,A -85,B 0,C 180,E1 23916.527,E2 23916.527} C_VEL
LIN {X 0,Y 529.913,Z 1062.851,A -85,B 0,C 180,E1 23914.997,E2 23914.997} C_VEL
LIN {X 0,Y 530.173,Z 1056.184,A -85,B 0,C 180,E1 23913.812,E2 23913.812} C_VEL
LIN {X 0,Y 530.486,Z 1048.287,A -85,B 0,C 180,E1 23912.686,E2 23912.686} C_VEL
LIN {X 0,Y 530.895,Z 1037.423,A -85,B 0,C 180,E1 23911.454,E2 23911.454} C_VEL
LIN {X 0,Y 531.234,Z 1026.612,A -85,B 0,C 180,E1 23910.501,E2 23910.501} C_VEL
LIN {X 0,Y 531.521,Z 1015.714,A -85,B 0,C 180,E1 23909.724,E2 23909.724} C_VEL
LIN {X 0,Y 531.807,Z 1002.658,A -85,B 0,C 180,E1 23908.991,E2 23908.991} C_VEL
LIN {X 0,Y 531.959,Z 987.834,A -85,B 0,C 180,E1 23908.401,E2 23908.401} C_VEL
LIN {X 0,Y 531.981,Z 975.252,A -85,B 0,C 180,E1 23908.06,E2 23908.06} C_VEL
LIN {X 0,Y 531.95,Z 953.396,A -85,B 0,C 180,E1 23907.71,E2 23907.71} C_VEL
LIN {X 0,Y 533.036,Z 856.533,A -85,B 0,C 180,E1 23906.304,E2 23906.304} C_VEL
LIN {X 0,Y 533.855,Z 841.052,A -85,B 0,C 180,E1 23905.639,E2 23905.639} C_VEL
LIN {X 0,Y 535.2,Z 780.103,A -85,B 0,C 180,E1 23902.92,E2 23902.92} C_VEL
LIN {X 0,Y 536.102,Z 781.31,A -85,B 0,C 180,E1 23902.754,E2 23902.754} C_VEL
LIN {X 0,Y 537.685,Z 781.196,A -85,B 0,C 180,E1 23902.548,E2 23902.548} C_VEL
LIN {X 0,Y 540.431,Z 778.707,A -85,B 0,C 180,E1 23902.27,E2 23902.27} C_VEL
LIN {X 0,Y 544.096,Z 772.998,A -85,B 0,C 180,E1 23901.985,E2 23901.985} C_VEL
LIN {X 0,Y 544.796,Z 772.069,A -85,B 0,C 180,E1 23901.926,E2 23901.926} C_VEL
LIN {X 0,Y 548.081,Z 770.377,A -85,B 0,C 180,E1 23901.563,E2 23901.563} C_VEL
LIN {X 0,Y 552.003,Z 766.221,A -85,B 0,C 180,E1 23901.206,E2 23901.206} C_VEL
LIN {X 0,Y 555.023,Z 761.8,A -85,B 0,C 180,E1 23900.977,E2 23900.977} C_VEL
LIN {X 0,Y 559.45,Z 758.649,A -85,B 0,C 180,E1 23900.544,E2 23900.544} C_VEL
LIN {X 0,Y 564.065,Z 753.294,A -85,B 0,C 180,E1 23900.164,E2 23900.164} C_VEL
LIN {X 0,Y 565.788,Z 751.087,A -85,B 0,C 180,E1 23900.029,E2 23900.029} C_VEL
LIN {X 0,Y 570.899,Z 746.974,A -85,B 0,C 180,E1 23899.574,E2 23899.574} C_VEL
LIN {X 0,Y 576.752,Z 740.215,A -85,B 0,C 180,E1 23899.121,E2 23899.121} C_VEL
LIN {X 0,Y 580.995,Z 737.005,A -85,B 0,C 180,E1 23898.76,E2 23898.76} C_VEL
LIN {X 0,Y 578.146,Z 782.095,A -85,B 0,C 180,E1 23897.929,E2 23897.929} C_VEL
LIN {X 0,Y 576.919,Z 789.729,A -85,B 0,C 180,E1 23897.861,E2 23897.861} C_VEL
LIN {X 0,Y 571.233,Z 809.032,A -85,B 0,C 180,E1 23897.9,E2 23897.9} C_VEL
LIN {X 0,Y 569.937,Z 816.635,A -85,B 0,C 180,E1 23897.81,E2 23897.81} C_VEL
LIN {X 0,Y 567.363,Z 845.633,A -85,B 0,C 180,E1 23897.063,E2 23897.063} C_VEL
LIN {X 0,Y 564.895,Z 868.937,A -85,B 0,C 180,E1 23896.309,E2 23896.309} C_VEL
LIN {X 0,Y 561.565,Z 897.237,A -85,B 0,C 180,E1 23895.199,E2 23895.199} C_VEL
LIN {X 0,Y 557.485,Z 930.047,A -85,B 0,C 180,E1 23893.673,E2 23893.673} C_VEL
LIN {X 0,Y 554.428,Z 953.413,A -85,B 0,C 180,E1 23892.416,E2 23892.416} C_VEL
LIN {X 0,Y 550.914,Z 978.44,A -85,B 0,C 180,E1 23890.867,E2 23890.867} C_VEL
LIN {X 0,Y 547.794,Z 998.225,A -85,B 0,C 180,E1 23889.436,E2 23889.436} C_VEL
LIN {X 0,Y 544.744,Z 1016.471,A -85,B 0,C 180,E1 23887.946,E2 23887.946} C_VEL
LIN {X 0,Y 541.284,Z 1036.48,A -85,B 0,C 180,E1 23886.106,E2 23886.106} C_VEL
LIN {X 0,Y 537.472,Z 1056.587,A -85,B 0,C 180,E1 23883.926,E2 23883.926} C_VEL
LIN {X 0,Y 533.834,Z 1075.636,A -85,B 0,C 180,E1 23881.544,E2 23881.544} C_VEL
LIN {X 0,Y 531.127,Z 1089.09,A -85,B 0,C 180,E1 23879.554,E2 23879.554} C_VEL
LIN {X 0,Y 528.536,Z 1102.24,A -85,B 0,C 180,E1 23877.369,E2 23877.369} C_VEL
LIN {X 0,Y 526.381,Z 1114.011,A -85,B 0,C 180,E1 23875.183,E2 23875.183} C_VEL
LIN {X 0,Y 524.627,Z 1124.554,A -85,B 0,C 180,E1 23872.992,E2 23872.992} C_VEL
LIN {X 0,Y 523.244,Z 1133.865,A -85,B 0,C 180,E1 23870.821,E2 23870.821} C_VEL
LIN {X 0,Y 522.098,Z 1142.527,A -85,B 0,C 180,E1 23868.538,E2 23868.538} C_VEL
LIN {X 0,Y 521.223,Z 1150.412,A -85,B 0,C 180,E1 23866.152,E2 23866.152} C_VEL
LIN {X 0,Y 520.615,Z 1157.51,A -85,B 0,C 180,E1 23863.633,E2 23863.633} C_VEL
LIN {X 0,Y 520.189,Z 1164.404,A -85,B 0,C 180,E1 23860.635,E2 23860.635} C_VEL
LIN {X 0,Y 519.987,Z 1169.464,A -85,B 0,C 180,E1 23857.626,E2 23857.626} C_VEL
LIN {X 0,Y 519.926,Z 1172.479,A -85,B 0,C 180,E1 23855.077,E2 23855.077} C_VEL
LIN {X 0,Y 519.907,Z 1174.238,A -85,B 0,C 180,E1 23852.647,E2 23852.647} C_VEL
LIN {X 0,Y 519.901,Z 1174.902,A -85,B 0,C 180,E1 23850.222,E2 23850.222} C_VEL
LIN {X 0,Y 519.91,Z 1174.474,A -85,B 0,C 180,E1 23847.797,E2 23847.797} C_VEL
LIN {X 0,Y 519.917,Z 1173.048,A -85,B 0,C 180,E1 23845.479,E2 23845.479} C_VEL
LIN {X 0,Y 519.957,Z 1170.615,A -85,B 0,C 180,E1 23843.154,E2 23843.154} C_VEL
LIN {X 0,Y 520.06,Z 1167.159,A -85,B 0,C 180,E1 23840.819,E2 23840.819} C_VEL
LIN {X 0,Y 520.283,Z 1162.408,A -85,B 0,C 180,E1 23838.36,E2 23838.36} C_VEL
LIN {X 0,Y 520.67,Z 1156.768,A -85,B 0,C 180,E1 23835.999,E2 23835.999} C_VEL
LIN {X 0,Y 521.266,Z 1149.992,A -85,B 0,C 180,E1 23833.624,E2 23833.624} C_VEL
LIN {X 0,Y 522.108,Z 1142.447,A -85,B 0,C 180,E1 23831.35,E2 23831.35} C_VEL
LIN {X 0,Y 523.254,Z 1133.768,A -85,B 0,C 180,E1 23829.065,E2 23829.065} C_VEL
LIN {X 0,Y 524.651,Z 1124.406,A -85,B 0,C 180,E1 23826.886,E2 23826.886} C_VEL
LIN {X 0,Y 526.398,Z 1113.878,A -85,B 0,C 180,E1 23824.7,E2 23824.7} C_VEL
LIN {X 0,Y 528.434,Z 1102.734,A -85,B 0,C 180,E1 23822.628,E2 23822.628} C_VEL
LIN {X 0,Y 530.868,Z 1090.346,A -85,B 0,C 180,E1 23820.557,E2 23820.557} C_VEL
LIN {X 0,Y 533.507,Z 1077.331,A -85,B 0,C 180,E1 23818.601,E2 23818.601} C_VEL
LIN {X 0,Y 536.705,Z 1060.706,A -85,B 0,C 180,E1 23816.465,E2 23816.465} C_VEL
LIN {X 0,Y 540.274,Z 1041.651,A -85,B 0,C 180,E1 23814.342,E2 23814.342} C_VEL
LIN {X 0,Y 543.232,Z 1025.165,A -85,B 0,C 180,E1 23812.733,E2 23812.733} C_VEL
LIN {X 0,Y 546.911,Z 1003.595,A -85,B 0,C 180,E1 23810.897,E2 23810.897} C_VEL
LIN {X 0,Y 549.849,Z 985.314,A -85,B 0,C 180,E1 23809.521,E2 23809.521} C_VEL
LIN {X 0,Y 552.656,Z 966.119,A -85,B 0,C 180,E1 23808.259,E2 23808.259} C_VEL
LIN {X 0,Y 555.999,Z 941.818,A -85,B 0,C 180,E1 23806.85,E2 23806.85} C_VEL
LIN {X 0,Y 559.045,Z 917.291,A -85,B 0,C 180,E1 23805.629,E2 23805.629} C_VEL
LIN {X 0,Y 562.66,Z 888.24,A -85,B 0,C 180,E1 23804.337,E2 23804.337} C_VEL
LIN {X 0,Y 565.352,Z 864.756,A -85,B 0,C 180,E1 23803.457,E2 23803.457} C_VEL
LIN {X 0,Y 568.134,Z 837.965,A -85,B 0,C 180,E1 23802.626,E2 23802.626} C_VEL
LIN {X 0,Y 570.229,Z 812.803,A -85,B 0,C 180,E1 23802.021,E2 23802.021} C_VEL
LIN {X 0,Y 581.369,Z 653.084,A -85,B 0,C 180,E1 23799.032,E2 23799.032} C_VEL
LIN {X 0,Y 588.697,Z 542.277,A -85,B 0,C 180,E1 23797.122,E2 23797.122} C_VEL
LIN {X 0,Y 593.658,Z 449.461,A -85,B 0,C 180,E1 23795.646,E2 23795.646} C_VEL
LIN {X 0,Y 594.213,Z 435.712,A -85,B 0,C 180,E1 23795.429,E2 23795.429} C_VEL
LIN {X 0,Y 583.471,Z 425.355,A -85,B 0,C 180,E1 23793.668,E2 23793.668} C_VEL
LIN {X 0,Y 575.075,Z 417.863,A -85,B 0,C 180,E1 23792.203,E2 23792.203} C_VEL
LIN {X 0,Y 568.176,Z 411.865,A -85,B 0,C 180,E1 23790.922,E2 23790.922} C_VEL
LIN {X 0,Y 563.423,Z 407.854,A -85,B 0,C 180,E1 23789.972,E2 23789.972} C_VEL
LIN {X 0,Y 562.355,Z 405.636,A -85,B 0,C 180,E1 23789.039,E2 23789.039} C_VEL
LIN {X 0,Y 559.887,Z 400.987,A -85,B 0,C 180,E1 23786.747,E2 23786.747} C_VEL
LIN {X 0,Y 557.743,Z 396.707,A -85,B 0,C 180,E1 23784.239,E2 23784.239} C_VEL
LIN {X 0,Y 554.814,Z 391.2,A -85,B 0,C 180,E1 23779.257,E2 23779.257} C_VEL
LIN {X 0,Y 553.49,Z 389.89,A -85,B 0,C 180,E1 23774.65,E2 23774.65} C_VEL
LIN {X 0,Y 554.123,Z 390.592,A -85,B 0,C 180,E1 23770.606,E2 23770.606} C_VEL
LIN {X 0,Y 555.153,Z 391.773,A -85,B 0,C 180,E1 23768.389,E2 23768.389} C_VEL
LIN {X 0,Y 558.013,Z 397.059,A -85,B 0,C 180,E1 23763.904,E2 23763.904} C_VEL
LIN {X 0,Y 560.418,Z 401.415,A -85,B 0,C 180,E1 23761.329,E2 23761.329} C_VEL
LIN {X 0,Y 563.501,Z 407.348,A -85,B 0,C 180,E1 23758.577,E2 23758.577} C_VEL
LIN {X 0,Y 566.151,Z 412.476,A -85,B 0,C 180,E1 23756.557,E2 23756.557} C_VEL
LIN {X 0,Y 568.66,Z 417.3,A -85,B 0,C 180,E1 23754.855,E2 23754.855} C_VEL
LIN {X 0,Y 572.792,Z 425.129,A -85,B 0,C 180,E1 23752.376,E2 23752.376} C_VEL
LIN {X 0,Y 577.533,Z 435.047,A -85,B 0,C 180,E1 23749.728,E2 23749.728} C_VEL
LIN {X 0,Y 582.779,Z 446.119,A -85,B 0,C 180,E1 23747.112,E2 23747.112} C_VEL
LIN {X 0,Y 587.92,Z 457.655,A -85,B 0,C 180,E1 23744.715,E2 23744.715} C_VEL
LIN {X 0,Y 588.056,Z 458.494,A -85,B 0,C 180,E1 23744.591,E2 23744.591} C_VEL
LIN {X 0,Y 582.132,Z 492.323,A -85,B 0,C 180,E1 23741.628,E2 23741.628} C_VEL
LIN {X 0,Y 576.268,Z 528.023,A -85,B 0,C 180,E1 23738.631,E2 23738.631} C_VEL
LIN {X 0,Y 570.335,Z 566.849,A -85,B 0,C 180,E1 23735.485,E2 23735.485} C_VEL
LIN {X 0,Y 565.66,Z 603.135,A -85,B 0,C 180,E1 23732.576,E2 23732.576} C_VEL
LIN {X 0,Y 565.216,Z 622.064,A -85,B 0,C 180,E1 23730.89,E2 23730.89} C_VEL
LIN {X 0,Y 566.757,Z 638.971,A -85,B 0,C 180,E1 23729.228,E2 23729.228} C_VEL
LIN {X 0,Y 569.985,Z 653.601,A -85,B 0,C 180,E1 23727.653,E2 23727.653} C_VEL
LIN {X 0,Y 575.047,Z 667.463,A -85,B 0,C 180,E1 23726.034,E2 23726.034} C_VEL
LIN {X 0,Y 582.548,Z 681.102,A -85,B 0,C 180,E1 23724.297,E2 23724.297} C_VEL
LIN {X 0,Y 590.703,Z 691.756,A -85,B 0,C 180,E1 23722.821,E2 23722.821} C_VEL
LIN {X 0,Y 601.687,Z 702.453,A -85,B 0,C 180,E1 23721.207,E2 23721.207} C_VEL
LIN {X 0,Y 605.158,Z 705.487,A -85,B 0,C 180,E1 23720.741,E2 23720.741} C_VEL
LIN {X 0,Y 594.84,Z 720.025,A -85,B 0,C 180,E1 23720.415,E2 23720.415} C_VEL
LIN {X 0,Y 587.666,Z 732.146,A -85,B 0,C 180,E1 23720.061,E2 23720.061} C_VEL
LIN {X 0,Y 583.956,Z 754.866,A -85,B 0,C 180,E1 23720.077,E2 23720.077} C_VEL
LIN {X 0,Y 582.147,Z 772.749,A -85,B 0,C 180,E1 23719.966,E2 23719.966} C_VEL
LIN {X 0,Y 580.383,Z 811.333,A -85,B 0,C 180,E1 23719.379,E2 23719.379} C_VEL
LIN {X 0,Y 577.508,Z 845.539,A -85,B 0,C 180,E1 23718.724,E2 23718.724} C_VEL
LIN {X 0,Y 574.331,Z 876.686,A -85,B 0,C 180,E1 23717.941,E2 23717.941} C_VEL
LIN {X 0,Y 570.924,Z 906.638,A -85,B 0,C 180,E1 23716.983,E2 23716.983} C_VEL
LIN {X 0,Y 567.373,Z 934.701,A -85,B 0,C 180,E1 23715.884,E2 23715.884} C_VEL
LIN {X 0,Y 563.587,Z 961.331,A -85,B 0,C 180,E1 23714.63,E2 23714.63} C_VEL
LIN {X 0,Y 559.783,Z 984.975,A -85,B 0,C 180,E1 23713.304,E2 23713.304} C_VEL
LIN {X 0,Y 555.653,Z 1007.377,A -85,B 0,C 180,E1 23711.818,E2 23711.818} C_VEL
LIN {X 0,Y 551.65,Z 1026.702,A -85,B 0,C 180,E1 23710.319,E2 23710.319} C_VEL
LIN {X 0,Y 547.555,Z 1045.787,A -85,B 0,C 180,E1 23708.645,E2 23708.645} C_VEL
LIN {X 0,Y 543.16,Z 1065.241,A -85,B 0,C 180,E1 23706.679,E2 23706.679} C_VEL
LIN {X 0,Y 538.325,Z 1086.048,A -85,B 0,C 180,E1 23704.247,E2 23704.247} C_VEL
LIN {X 0,Y 534.294,Z 1104.125,A -85,B 0,C 180,E1 23701.851,E2 23701.851} C_VEL
LIN {X 0,Y 530.483,Z 1122.278,A -85,B 0,C 180,E1 23699.095,E2 23699.095} C_VEL
LIN {X 0,Y 527.553,Z 1137.707,A -85,B 0,C 180,E1 23696.447,E2 23696.447} C_VEL
LIN {X 0,Y 525.042,Z 1152.214,A -85,B 0,C 180,E1 23693.572,E2 23693.572} C_VEL
LIN {X 0,Y 523.219,Z 1164.118,A -85,B 0,C 180,E1 23690.819,E2 23690.819} C_VEL
LIN {X 0,Y 521.852,Z 1174.735,A -85,B 0,C 180,E1 23687.966,E2 23687.966} C_VEL
LIN {X 0,Y 520.924,Z 1183.954,A -85,B 0,C 180,E1 23685.017,E2 23685.017} C_VEL
LIN {X 0,Y 520.363,Z 1191.145,A -85,B 0,C 180,E1 23682.201,E2 23682.201} C_VEL
LIN {X 0,Y 520.079,Z 1196.733,A -85,B 0,C 180,E1 23679.404,E2 23679.404} C_VEL
LIN {X 0,Y 519.957,Z 1200.907,A -85,B 0,C 180,E1 23676.624,E2 23676.624} C_VEL
LIN {X 0,Y 519.914,Z 1203.585,A -85,B 0,C 180,E1 23673.858,E2 23673.858} C_VEL
LIN {X 0,Y 519.913,Z 1204.828,A -85,B 0,C 180,E1 23671.101,E2 23671.101} C_VEL
LIN {X 0,Y 519.909,Z 1204.749,A -85,B 0,C 180,E1 23668.456,E2 23668.456} C_VEL
LIN {X 0,Y 519.918,Z 1203.231,A -85,B 0,C 180,E1 23665.697,E2 23665.697} C_VEL
LIN {X 0,Y 519.97,Z 1200.261,A -85,B 0,C 180,E1 23662.867,E2 23662.867} C_VEL
LIN {X 0,Y 520.114,Z 1195.946,A -85,B 0,C 180,E1 23660.147,E2 23660.147} C_VEL
LIN {X 0,Y 520.447,Z 1189.79,A -85,B 0,C 180,E1 23657.235,E2 23657.235} C_VEL
LIN {X 0,Y 521.065,Z 1182.328,A -85,B 0,C 180,E1 23654.415,E2 23654.415} C_VEL
LIN {X 0,Y 522.111,Z 1172.705,A -85,B 0,C 180,E1 23651.437,E2 23651.437} C_VEL
LIN {X 0,Y 523.547,Z 1161.757,A -85,B 0,C 180,E1 23648.605,E2 23648.605} C_VEL
LIN {X 0,Y 525.628,Z 1148.545,A -85,B 0,C 180,E1 23645.671,E2 23645.671} C_VEL
LIN {X 0,Y 528.24,Z 1133.836,A -85,B 0,C 180,E1 23642.858,E2 23642.858} C_VEL
LIN {X 0,Y 531.085,Z 1119.364,A -85,B 0,C 180,E1 23640.438,E2 23640.438} C_VEL
LIN {X 0,Y 534.817,Z 1101.566,A -85,B 0,C 180,E1 23637.802,E2 23637.802} C_VEL
LIN {X 0,Y 538.544,Z 1085.127,A -85,B 0,C 180,E1 23635.637,E2 23635.637} C_VEL
LIN {X 0,Y 543.498,Z 1063.728,A -85,B 0,C 180,E1 23633.158,E2 23633.158} C_VEL
LIN {X 0,Y 547.958,Z 1044.005,A -85,B 0,C 180,E1 23631.185,E2 23631.185} C_VEL
LIN {X 0,Y 552.74,Z 1021.985,A -85,B 0,C 180,E1 23629.285,E2 23629.285} C_VEL
LIN {X 0,Y 556.866,Z 1000.952,A -85,B 0,C 180,E1 23627.737,E2 23627.737} C_VEL
LIN {X 0,Y 560.755,Z 979.438,A -85,B 0,C 180,E1 23626.364,E2 23626.364} C_VEL
LIN {X 0,Y 564.436,Z 955.901,A -85,B 0,C 180,E1 23625.094,E2 23625.094} C_VEL
LIN {X 0,Y 568.187,Z 928.58,A -85,B 0,C 180,E1 23623.856,E2 23623.856} C_VEL
LIN {X 0,Y 571.755,Z 899.618,A -85,B 0,C 180,E1 23622.771,E2 23622.771} C_VEL
LIN {X 0,Y 575.137,Z 869.294,A -85,B 0,C 180,E1 23621.854,E2 23621.854} C_VEL
LIN {X 0,Y 578.171,Z 838.712,A -85,B 0,C 180,E1 23621.13,E2 23621.13} C_VEL
LIN {X 0,Y 580.78,Z 804.44,A -85,B 0,C 180,E1 23620.507,E2 23620.507} C_VEL
LIN {X 0,Y 583.109,Z 745.707,A -85,B 0,C 180,E1 23619.659,E2 23619.659} C_VEL
LIN {X 0,Y 584.483,Z 718.039,A -85,B 0,C 180,E1 23619.263,E2 23619.263} C_VEL
LIN {X 0,Y 590.361,Z 659.419,A -85,B 0,C 180,E1 23618.276,E2 23618.276} C_VEL
LIN {X 0,Y 594.716,Z 616.335,A -85,B 0,C 180,E1 23617.555,E2 23617.555} C_VEL
LIN {X 0,Y 596.826,Z 598.038,A -85,B 0,C 180,E1 23617.279,E2 23617.279} C_VEL
LIN {X 0,Y 599.868,Z 567.606,A -85,B 0,C 180,E1 23616.766,E2 23616.766} C_VEL
LIN {X 0,Y 603.303,Z 540.205,A -85,B 0,C 180,E1 23616.387,E2 23616.387} C_VEL
LIN {X 0,Y 605.974,Z 512.789,A -85,B 0,C 180,E1 23615.916,E2 23615.916} C_VEL
LIN {X 0,Y 610.625,Z 477.551,A -85,B 0,C 180,E1 23615.459,E2 23615.459} C_VEL
LIN {X 0,Y 611.832,Z 462.005,A -85,B 0,C 180,E1 23615.155,E2 23615.155} C_VEL
LIN {X 0,Y 595.738,Z 436.559,A -85,B 0,C 180,E1 23612.258,E2 23612.258} C_VEL
LIN {X 0,Y 584.049,Z 419.081,A -85,B 0,C 180,E1 23609.937,E2 23609.937} C_VEL
LIN {X 0,Y 573.336,Z 403.94,A -85,B 0,C 180,E1 23607.611,E2 23607.611} C_VEL
LIN {X 0,Y 564.609,Z 392.375,A -85,B 0,C 180,E1 23605.545,E2 23605.545} C_VEL
LIN {X 0,Y 560.7,Z 387.218,A -85,B 0,C 180,E1 23604.551,E2 23604.551} C_VEL
LIN {X 0,Y 556.744,Z 382.068,A -85,B 0,C 180,E1 23603.497,E2 23603.497} C_VEL
LIN {X 0,Y 552.592,Z 376.77,A -85,B 0,C 180,E1 23602.333,E2 23602.333} C_VEL
LIN {X 0,Y 549.08,Z 372.522,A -85,B 0,C 180,E1 23601.303,E2 23601.303} C_VEL
LIN {X 0,Y 547.97,Z 370.987,A -85,B 0,C 180,E1 23600.956,E2 23600.956} C_VEL
LIN {X 0,Y 544.615,Z 367.207,A -85,B 0,C 180,E1 23599.912,E2 23599.912} C_VEL
LIN {X 0,Y 543.158,Z 364.982,A -85,B 0,C 180,E1 23599.407,E2 23599.407} C_VEL
LIN {X 0,Y 539.955,Z 361.868,A -85,B 0,C 180,E1 23598.349,E2 23598.349} C_VEL
LIN {X 0,Y 538.103,Z 358.796,A -85,B 0,C 180,E1 23597.631,E2 23597.631} C_VEL
LIN {X 0,Y 535.54,Z 356.99,A -85,B 0,C 180,E1 23596.738,E2 23596.738} C_VEL
LIN {X 0,Y 534.692,Z 358.124,A -85,B 0,C 180,E1 23596.542,E2 23596.542} C_VEL
LIN {X 0,Y 532.681,Z 362.228,A -85,B 0,C 180,E1 23596.158,E2 23596.158} C_VEL
LIN {X 0,Y 531.396,Z 363.747,A -85,B 0,C 180,E1 23595.833,E2 23595.833} C_VEL
LIN {X 0,Y 531.013,Z 364.012,A -85,B 0,C 180,E1 23595.698,E2 23595.698} C_VEL
LIN {X 0,Y 530.501,Z 441.862,A -85,B 0,C 180,E1 23592.823,E2 23592.823} C_VEL
LIN {X 0,Y 530.414,Z 521.513,A -85,B 0,C 180,E1 23589.753,E2 23589.753} C_VEL
LIN {X 0,Y 529.92,Z 598.769,A -85,B 0,C 180,E1 23586.691,E2 23586.691} C_VEL
LIN {X 0,Y 529.039,Z 676.72,A -85,B 0,C 180,E1 23583.522,E2 23583.522} C_VEL
LIN {X 0,Y 527.83,Z 754.899,A -85,B 0,C 180,E1 23580.271,E2 23580.271} C_VEL
LIN {X 0,Y 526.513,Z 834.496,A -85,B 0,C 180,E1 23576.897,E2 23576.897} C_VEL
LIN {X 0,Y 525.82,Z 854.578,A -85,B 0,C 180,E1 23576.047,E2 23576.047} C_VEL
LIN {X 0,Y 525.04,Z 865.355,A -85,B 0,C 180,E1 23575.635,E2 23575.635} C_VEL
LIN {X 0,Y 524.052,Z 973.863,A -85,B 0,C 180,E1 23574.012,E2 23574.012} C_VEL
LIN {X 0,Y 524.134,Z 989.577,A -85,B 0,C 180,E1 23573.644,E2 23573.644} C_VEL
LIN {X 0,Y 524.097,Z 1001.604,A -85,B 0,C 180,E1 23573.207,E2 23573.207} C_VEL
LIN {X 0,Y 523.962,Z 1012.975,A -85,B 0,C 180,E1 23572.654,E2 23572.654} C_VEL
LIN {X 0,Y 523.73,Z 1025.341,A -85,B 0,C 180,E1 23571.878,E2 23571.878} C_VEL
LIN {X 0,Y 523.401,Z 1036.75,A -85,B 0,C 180,E1 23570.932,E2 23570.932} C_VEL
LIN {X 0,Y 523.109,Z 1044.97,A -85,B 0,C 180,E1 23570.094,E2 23570.094} C_VEL
LIN {X 0,Y 522.781,Z 1053.081,A -85,B 0,C 180,E1 23569.085,E2 23569.085} C_VEL
LIN {X 0,Y 522.492,Z 1059.721,A -85,B 0,C 180,E1 23568.072,E2 23568.072} C_VEL
LIN {X 0,Y 522.212,Z 1065.685,A -85,B 0,C 180,E1 23566.942,E2 23566.942} C_VEL
LIN {X 0,Y 521.953,Z 1071.23,A -85,B 0,C 180,E1 23565.579,E2 23565.579} C_VEL
LIN {X 0,Y 521.736,Z 1075.29,A -85,B 0,C 180,E1 23564.094,E2 23564.094} C_VEL
LIN {X 0,Y 521.61,Z 1077.525,A -85,B 0,C 180,E1 23562.715,E2 23562.715} C_VEL
LIN {X 0,Y 521.542,Z 1078.371,A -85,B 0,C 180,E1 23561.443,E2 23561.443} C_VEL
LIN {X 0,Y 521.524,Z 1078.049,A -85,B 0,C 180,E1 23560.162,E2 23560.162} C_VEL
LIN {X 0,Y 521.566,Z 1076.201,A -85,B 0,C 180,E1 23558.639,E2 23558.639} C_VEL
LIN {X 0,Y 521.69,Z 1072.469,A -85,B 0,C 180,E1 23557.103,E2 23557.103} C_VEL
LIN {X 0,Y 521.853,Z 1067.802,A -85,B 0,C 180,E1 23555.789,E2 23555.789} C_VEL
LIN {X 0,Y 522.077,Z 1062.238,A -85,B 0,C 180,E1 23554.595,E2 23554.595} C_VEL
LIN {X 0,Y 522.415,Z 1054.398,A -85,B 0,C 180,E1 23553.27,E2 23553.27} C_VEL
LIN {X 0,Y 522.802,Z 1044.548,A -85,B 0,C 180,E1 23551.996,E2 23551.996} C_VEL
LIN {X 0,Y 523.151,Z 1035.145,A -85,B 0,C 180,E1 23551.019,E2 23551.019} C_VEL
LIN {X 0,Y 523.483,Z 1024.672,A -85,B 0,C 180,E1 23550.133,E2 23550.133} C_VEL
LIN {X 0,Y 523.843,Z 1011.127,A -85,B 0,C 180,E1 23549.233,E2 23549.233} C_VEL
LIN {X 0,Y 524.056,Z 998.53,A -85,B 0,C 180,E1 23548.609,E2 23548.609} C_VEL
LIN {X 0,Y 524.16,Z 986.385,A -85,B 0,C 180,E1 23548.159,E2 23548.159} C_VEL
LIN {X 0,Y 524.18,Z 972.504,A -85,B 0,C 180,E1 23547.809,E2 23547.809} C_VEL
LIN {X 0,Y 525.294,Z 857.231,A -85,B 0,C 180,E1 23546.092,E2 23546.092} C_VEL
LIN {X 0,Y 526.151,Z 841.452,A -85,B 0,C 180,E1 23545.407,E2 23545.407} C_VEL
LIN {X 0,Y 527.17,Z 797.177,A -85,B 0,C 180,E1 23543.413,E2 23543.413} C_VEL
LIN {X 0,Y 528.045,Z 798.344,A -85,B 0,C 180,E1 23543.247,E2 23543.247} C_VEL
LIN {X 0,Y 529.62,Z 798.246,A -85,B 0,C 180,E1 23543.036,E2 23543.036} C_VEL
LIN {X 0,Y 532.361,Z 795.718,A -85,B 0,C 180,E1 23542.753,E2 23542.753} C_VEL
LIN {X 0,Y 536.154,Z 789.792,A -85,B 0,C 180,E1 23542.455,E2 23542.455} C_VEL
LIN {X 0,Y 536.728,Z 789.136,A -85,B 0,C 180,E1 23542.402,E2 23542.402} C_VEL
LIN {X 0,Y 540.004,Z 787.442,A -85,B 0,C 180,E1 23542.033,E2 23542.033} C_VEL
LIN {X 0,Y 543.828,Z 783.425,A -85,B 0,C 180,E1 23541.678,E2 23541.678} C_VEL
LIN {X 0,Y 546.937,Z 778.896,A -85,B 0,C 180,E1 23541.435,E2 23541.435} C_VEL
LIN {X 0,Y 551.303,Z 775.763,A -85,B 0,C 180,E1 23540.998,E2 23540.998} C_VEL
LIN {X 0,Y 555.963,Z 770.324,A -85,B 0,C 180,E1 23540.606,E2 23540.606} C_VEL
LIN {X 0,Y 557.702,Z 768.086,A -85,B 0,C 180,E1 23540.471,E2 23540.471} C_VEL
LIN {X 0,Y 562.798,Z 763.929,A -85,B 0,C 180,E1 23540.006,E2 23540.006} C_VEL
LIN {X 0,Y 568.437,Z 757.329,A -85,B 0,C 180,E1 23539.561,E2 23539.561} C_VEL
LIN {X 0,Y 574.251,Z 752.347,A -85,B 0,C 180,E1 23539.07,E2 23539.07} C_VEL
LIN {X 0,Y 574.437,Z 752.356,A -85,B 0,C 180,E1 23539.051,E2 23539.051} C_VEL
LIN {X 0,Y 569.937,Z 816.635,A -85,B 0,C 180,E1 23537.81,E2 23537.81} C_VEL
LIN {X 0,Y 568.004,Z 826.375,A -85,B 0,C 180,E1 23537.698,E2 23537.698} C_VEL
LIN {X 0,Y 562.395,Z 843.346,A -85,B 0,C 180,E1 23537.63,E2 23537.63} C_VEL
LIN {X 0,Y 560.932,Z 850.786,A -85,B 0,C 180,E1 23537.463,E2 23537.463} C_VEL
LIN {X 0,Y 558.384,Z 873.332,A -85,B 0,C 180,E1 23536.699,E2 23536.699} C_VEL
LIN {X 0,Y 554.922,Z 900.144,A -85,B 0,C 180,E1 23535.598,E2 23535.598} C_VEL
LIN {X 0,Y 551.642,Z 923.478,A -85,B 0,C 180,E1 23534.468,E2 23534.468} C_VEL
LIN {X 0,Y 546.76,Z 957.039,A -85,B 0,C 180,E1 23532.582,E2 23532.582} C_VEL
LIN {X 0,Y 543.034,Z 982.333,A -85,B 0,C 180,E1 23530.959,E2 23530.959} C_VEL
LIN {X 0,Y 539.904,Z 1002.053,A -85,B 0,C 180,E1 23529.507,E2 23529.507} C_VEL
LIN {X 0,Y 537.315,Z 1017.225,A -85,B 0,C 180,E1 23528.251,E2 23528.251} C_VEL
LIN {X 0,Y 533.727,Z 1037.457,A -85,B 0,C 180,E1 23526.366,E2 23526.366} C_VEL
LIN {X 0,Y 530.15,Z 1056.344,A -85,B 0,C 180,E1 23524.329,E2 23524.329} C_VEL
LIN {X 0,Y 527.013,Z 1072.348,A -85,B 0,C 180,E1 23522.347,E2 23522.347} C_VEL
LIN {X 0,Y 523.787,Z 1088.86,A -85,B 0,C 180,E1 23520.011,E2 23520.011} C_VEL
LIN {X 0,Y 521.479,Z 1100.459,A -85,B 0,C 180,E1 23518.114,E2 23518.114} C_VEL
LIN {X 0,Y 519.038,Z 1112.848,A -85,B 0,C 180,E1 23515.81,E2 23515.81} C_VEL
LIN {X 0,Y 517.137,Z 1123.533,A -85,B 0,C 180,E1 23513.582,E2 23513.582} C_VEL
LIN {X 0,Y 515.615,Z 1132.941,A -85,B 0,C 180,E1 23511.382,E2 23511.382} C_VEL
LIN {X 0,Y 514.368,Z 1141.715,A -85,B 0,C 180,E1 23509.062,E2 23509.062} C_VEL
LIN {X 0,Y 513.453,Z 1149.354,A -85,B 0,C 180,E1 23506.752,E2 23506.752} C_VEL
LIN {X 0,Y 512.796,Z 1155.921,A -85,B 0,C 180,E1 23504.454,E2 23504.454} C_VEL
LIN {X 0,Y 512.363,Z 1161.57,A -85,B 0,C 180,E1 23502.117,E2 23502.117} C_VEL
LIN {X 0,Y 512.113,Z 1166.207,A -85,B 0,C 180,E1 23499.781,E2 23499.781} C_VEL
LIN {X 0,Y 511.986,Z 1169.903,A -85,B 0,C 180,E1 23497.407,E2 23497.407} C_VEL
LIN {X 0,Y 511.927,Z 1172.576,A -85,B 0,C 180,E1 23495.041,E2 23495.041} C_VEL
LIN {X 0,Y 511.908,Z 1174.235,A -85,B 0,C 180,E1 23492.688,E2 23492.688} C_VEL
LIN {X 0,Y 511.901,Z 1174.899,A -85,B 0,C 180,E1 23490.225,E2 23490.225} C_VEL
LIN {X 0,Y 511.909,Z 1174.47,A -85,B 0,C 180,E1 23487.763,E2 23487.763} C_VEL
LIN {X 0,Y 511.917,Z 1173.044,A -85,B 0,C 180,E1 23485.408,E2 23485.408} C_VEL
LIN {X 0,Y 511.959,Z 1170.611,A -85,B 0,C 180,E1 23483.046,E2 23483.046} C_VEL
LIN {X 0,Y 512.073,Z 1167.155,A -85,B 0,C 180,E1 23480.675,E2 23480.675} C_VEL
LIN {X 0,Y 512.318,Z 1162.403,A -85,B 0,C 180,E1 23478.176,E2 23478.176} C_VEL
LIN {X 0,Y 512.735,Z 1156.679,A -85,B 0,C 180,E1 23475.745,E2 23475.745} C_VEL
LIN {X 0,Y 513.379,Z 1149.989,A -85,B 0,C 180,E1 23473.365,E2 23473.365} C_VEL
LIN {X 0,Y 514.272,Z 1142.443,A -85,B 0,C 180,E1 23471.055,E2 23471.055} C_VEL
LIN {X 0,Y 515.488,Z 1133.765,A -85,B 0,C 180,E1 23468.734,E2 23468.734} C_VEL
LIN {X 0,Y 517.044,Z 1124.042,A -85,B 0,C 180,E1 23466.442,E2 23466.442} C_VEL
LIN {X 0,Y 518.952,Z 1113.29,A -85,B 0,C 180,E1 23464.188,E2 23464.188} C_VEL
LIN {X 0,Y 521.412,Z 1100.782,A -85,B 0,C 180,E1 23461.854,E2 23461.854} C_VEL
LIN {X 0,Y 523.85,Z 1088.508,A -85,B 0,C 180,E1 23459.844,E2 23459.844} C_VEL
LIN {X 0,Y 527.369,Z 1070.581,A -85,B 0,C 180,E1 23457.334,E2 23457.334} C_VEL
LIN {X 0,Y 530.609,Z 1054.052,A -85,B 0,C 180,E1 23455.315,E2 23455.315} C_VEL
LIN {X 0,Y 534.42,Z 1033.429,A -85,B 0,C 180,E1 23453.158,E2 23453.158} C_VEL
LIN {X 0,Y 537.518,Z 1015.963,A -85,B 0,C 180,E1 23451.55,E2 23451.55} C_VEL
LIN {X 0,Y 540.099,Z 1000.789,A -85,B 0,C 180,E1 23450.307,E2 23450.307} C_VEL
LIN {X 0,Y 543.115,Z 981.73,A -85,B 0,C 180,E1 23448.912,E2 23448.912} C_VEL
LIN {X 0,Y 546.847,Z 956.314,A -85,B 0,C 180,E1 23447.287,E2 23447.287} C_VEL
LIN {X 0,Y 551.605,Z 923.692,A -85,B 0,C 180,E1 23445.454,E2 23445.454} C_VEL
LIN {X 0,Y 555.047,Z 899.241,A -85,B 0,C 180,E1 23444.271,E2 23444.271} C_VEL
LIN {X 0,Y 558.545,Z 871.871,A -85,B 0,C 180,E1 23443.159,E2 23443.159} C_VEL
LIN {X 0,Y 561.062,Z 849.627,A -85,B 0,C 180,E1 23442.411,E2 23442.411} C_VEL
LIN {X 0,Y 563.641,Z 823.532,A -85,B 0,C 180,E1 23441.69,E2 23441.69} C_VEL
LIN {X 0,Y 566.982,Z 779.46,A -85,B 0,C 180,E1 23440.793,E2 23440.793} C_VEL
LIN {X 0,Y 577.779,Z 632.856,A -85,B 0,C 180,E1 23438.05,E2 23438.05} C_VEL
LIN {X 0,Y 584.602,Z 531.569,A -85,B 0,C 180,E1 23436.311,E2 23436.311} C_VEL
LIN {X 0,Y 589.287,Z 444.34,A -85,B 0,C 180,E1 23434.93,E2 23434.93} C_VEL
LIN {X 0,Y 589.406,Z 440.773,A -85,B 0,C 180,E1 23434.869,E2 23434.869} C_VEL
LIN {X 0,Y 578.567,Z 430.515,A -85,B 0,C 180,E1 23433.042,E2 23433.042} C_VEL
LIN {X 0,Y 572.474,Z 425.034,A -85,B 0,C 180,E1 23431.953,E2 23431.953} C_VEL
LIN {X 0,Y 565.631,Z 419.052,A -85,B 0,C 180,E1 23430.664,E2 23430.664} C_VEL
LIN {X 0,Y 558.216,Z 412.612,A -85,B 0,C 180,E1 23429.158,E2 23429.158} C_VEL
LIN {X 0,Y 555.464,Z 407.599,A -85,B 0,C 180,E1 23426.63,E2 23426.63} C_VEL
LIN {X 0,Y 553.099,Z 402.9,A -85,B 0,C 180,E1 23423.775,E2 23423.775} C_VEL
LIN {X 0,Y 550.57,Z 397.976,A -85,B 0,C 180,E1 23419.191,E2 23419.191} C_VEL
LIN {X 0,Y 549.3,Z 396.705,A -85,B 0,C 180,E1 23414.656,E2 23414.656} C_VEL
LIN {X 0,Y 549.939,Z 397.415,A -85,B 0,C 180,E1 23410.582,E2 23410.582} C_VEL
LIN {X 0,Y 550.918,Z 398.532,A -85,B 0,C 180,E1 23408.454,E2 23408.454} C_VEL
LIN {X 0,Y 553.723,Z 403.859,A -85,B 0,C 180,E1 23403.935,E2 23403.935} C_VEL
LIN {X 0,Y 556.387,Z 408.897,A -85,B 0,C 180,E1 23401.03,E2 23401.03} C_VEL
LIN {X 0,Y 559.072,Z 414,A -85,B 0,C 180,E1 23398.65,E2 23398.65} C_VEL
LIN {X 0,Y 561.67,Z 419.093,A -85,B 0,C 180,E1 23396.632,E2 23396.632} C_VEL
LIN {X 0,Y 564.15,Z 423.932,A -85,B 0,C 180,E1 23394.916,E2 23394.916} C_VEL
LIN {X 0,Y 568.078,Z 431.449,A -85,B 0,C 180,E1 23392.516,E2 23392.516} C_VEL
LIN {X 0,Y 572.756,Z 441.373,A -85,B 0,C 180,E1 23389.844,E2 23389.844} C_VEL
LIN {X 0,Y 577.743,Z 452.029,A -85,B 0,C 180,E1 23387.303,E2 23387.303} C_VEL
LIN {X 0,Y 582.612,Z 463.062,A -85,B 0,C 180,E1 23384.98,E2 23384.98} C_VEL
LIN {X 0,Y 576.618,Z 496.009,A -85,B 0,C 180,E1 23382.073,E2 23382.073} C_VEL
LIN {X 0,Y 570.505,Z 531.744,A -85,B 0,C 180,E1 23379.051,E2 23379.051} C_VEL
LIN {X 0,Y 564.275,Z 570.848,A -85,B 0,C 180,E1 23375.859,E2 23375.859} C_VEL
LIN {X 0,Y 559.602,Z 605.325,A -85,B 0,C 180,E1 23373.071,E2 23373.071} C_VEL
LIN {X 0,Y 558.939,Z 624.509,A -85,B 0,C 180,E1 23371.352,E2 23371.352} C_VEL
LIN {X 0,Y 560.255,Z 641.591,A -85,B 0,C 180,E1 23369.664,E2 23369.664} C_VEL
LIN {X 0,Y 563.312,Z 656.605,A -85,B 0,C 180,E1 23368.041,E2 23368.041} C_VEL
LIN {X 0,Y 568.325,Z 671.067,A -85,B 0,C 180,E1 23366.344,E2 23366.344} C_VEL
LIN {X 0,Y 575.34,Z 684.421,A -85,B 0,C 180,E1 23364.639,E2 23364.639} C_VEL
LIN {X 0,Y 583.77,Z 695.952,A -85,B 0,C 180,E1 23363.044,E2 23363.044} C_VEL
LIN {X 0,Y 594.58,Z 706.874,A -85,B 0,C 180,E1 23361.398,E2 23361.398} C_VEL
LIN {X 0,Y 596.085,Z 708.375,A -85,B 0,C 180,E1 23361.178,E2 23361.178} C_VEL
LIN {X 0,Y 586.296,Z 722.926,A -85,B 0,C 180,E1 23360.813,E2 23360.813} C_VEL
LIN {X 0,Y 583.15,Z 728.492,A -85,B 0,C 180,E1 23360.659,E2 23360.659} C_VEL
LIN {X 0,Y 578.948,Z 753.905,A -85,B 0,C 180,E1 23360.687,E2 23360.687} C_VEL
LIN {X 0,Y 577.016,Z 772.76,A -85,B 0,C 180,E1 23360.574,E2 23360.574} C_VEL
LIN {X 0,Y 575.175,Z 809.464,A -85,B 0,C 180,E1 23360.006,E2 23360.006} C_VEL
LIN {X 0,Y 572.127,Z 844.332,A -85,B 0,C 180,E1 23359.333,E2 23359.333} C_VEL
LIN {X 0,Y 568.815,Z 875.33,A -85,B 0,C 180,E1 23358.554,E2 23358.554} C_VEL
LIN {X 0,Y 565.274,Z 905.223,A -85,B 0,C 180,E1 23357.601,E2 23357.601} C_VEL
LIN {X 0,Y 561.623,Z 933.25,A -85,B 0,C 180,E1 23356.507,E2 23356.507} C_VEL
LIN {X 0,Y 557.69,Z 960.612,A -85,B 0,C 180,E1 23355.232,E2 23355.232} C_VEL
LIN {X 0,Y 553.659,Z 985.917,A -85,B 0,C 180,E1 23353.833,E2 23353.833} C_VEL
LIN {X 0,Y 549.711,Z 1008,A -85,B 0,C 180,E1 23352.397,E2 23352.397} C_VEL
LIN {X 0,Y 545.869,Z 1026.572,A -85,B 0,C 180,E1 23350.975,E2 23350.975} C_VEL
LIN {X 0,Y 541.675,Z 1045.256,A -85,B 0,C 180,E1 23349.336,E2 23349.336} C_VEL
LIN {X 0,Y 537.131,Z 1064.04,A -85,B 0,C 180,E1 23347.428,E2 23347.428} C_VEL
LIN {X 0,Y 532.457,Z 1083.174,A -85,B 0,C 180,E1 23345.203,E2 23345.203} C_VEL
LIN {X 0,Y 527.616,Z 1102.83,A -85,B 0,C 180,E1 23342.56,E2 23342.56} C_VEL
LIN {X 0,Y 523.795,Z 1119.57,A -85,B 0,C 180,E1 23340.007,E2 23340.007} C_VEL
LIN {X 0,Y 520.166,Z 1137.099,A -85,B 0,C 180,E1 23336.976,E2 23336.976} C_VEL
LIN {X 0,Y 517.481,Z 1151.665,A -85,B 0,C 180,E1 23334.059,E2 23334.059} C_VEL
LIN {X 0,Y 515.513,Z 1163.649,A -85,B 0,C 180,E1 23331.265,E2 23331.265} C_VEL
LIN {X 0,Y 514.001,Z 1174.733,A -85,B 0,C 180,E1 23328.25,E2 23328.25} C_VEL
LIN {X 0,Y 513,Z 1183.978,A -85,B 0,C 180,E1 23325.245,E2 23325.245} C_VEL
LIN {X 0,Y 512.397,Z 1191.145,A -85,B 0,C 180,E1 23322.394,E2 23322.394} C_VEL
LIN {X 0,Y 512.094,Z 1196.732,A -85,B 0,C 180,E1 23319.552,E2 23319.552} C_VEL
LIN {X 0,Y 511.958,Z 1200.907,A -85,B 0,C 180,E1 23316.728,E2 23316.728} C_VEL
LIN {X 0,Y 511.916,Z 1203.496,A -85,B 0,C 180,E1 23314.031,E2 23314.031} C_VEL
LIN {X 0,Y 511.913,Z 1204.828,A -85,B 0,C 180,E1 23311.118,E2 23311.118} C_VEL
LIN {X 0,Y 511.909,Z 1204.751,A -85,B 0,C 180,E1 23308.432,E2 23308.432} C_VEL
LIN {X 0,Y 511.918,Z 1203.229,A -85,B 0,C 180,E1 23305.63,E2 23305.63} C_VEL
LIN {X 0,Y 511.976,Z 1200.333,A -85,B 0,C 180,E1 23302.807,E2 23302.807} C_VEL
LIN {X 0,Y 512.13,Z 1195.945,A -85,B 0,C 180,E1 23299.992,E2 23299.992} C_VEL
LIN {X 0,Y 512.496,Z 1189.788,A -85,B 0,C 180,E1 23297.033,E2 23297.033} C_VEL
LIN {X 0,Y 513.144,Z 1182.327,A -85,B 0,C 180,E1 23294.168,E2 23294.168} C_VEL
LIN {X 0,Y 514.26,Z 1172.789,A -85,B 0,C 180,E1 23291.169,E2 23291.169} C_VEL
LIN {X 0,Y 515.812,Z 1161.757,A -85,B 0,C 180,E1 23288.268,E2 23288.268} C_VEL
LIN {X 0,Y 517.964,Z 1148.856,A -85,B 0,C 180,E1 23285.355,E2 23285.355} C_VEL
LIN {X 0,Y 520.665,Z 1134.493,A -85,B 0,C 180,E1 23282.554,E2 23282.554} C_VEL
LIN {X 0,Y 524.607,Z 1116.027,A -85,B 0,C 180,E1 23279.409,E2 23279.409} C_VEL
LIN {X 0,Y 528.608,Z 1098.72,A -85,B 0,C 180,E1 23276.861,E2 23276.861} C_VEL
LIN {X 0,Y 533.367,Z 1079.449,A -85,B 0,C 180,E1 23274.335,E2 23274.335} C_VEL
LIN {X 0,Y 538.173,Z 1059.771,A -85,B 0,C 180,E1 23272.116,E2 23272.116} C_VEL
LIN {X 0,Y 542.741,Z 1040.969,A -85,B 0,C 180,E1 23270.261,E2 23270.261} C_VEL
LIN {X 0,Y 546.782,Z 1022.357,A -85,B 0,C 180,E1 23268.688,E2 23268.688} C_VEL
LIN {X 0,Y 550.091,Z 1005.772,A -85,B 0,C 180,E1 23267.453,E2 23267.453} C_VEL
LIN {X 0,Y 553.832,Z 984.973,A -85,B 0,C 180,E1 23266.109,E2 23266.109} C_VEL
LIN {X 0,Y 557.871,Z 959.495,A -85,B 0,C 180,E1 23264.711,E2 23264.711} C_VEL
LIN {X 0,Y 561.814,Z 931.971,A -85,B 0,C 180,E1 23263.435,E2 23263.435} C_VEL
LIN {X 0,Y 565.575,Z 902.974,A -85,B 0,C 180,E1 23262.316,E2 23262.316} C_VEL
LIN {X 0,Y 569.096,Z 872.989,A -85,B 0,C 180,E1 23261.379,E2 23261.379} C_VEL
LIN {X 0,Y 572.357,Z 842.074,A -85,B 0,C 180,E1 23260.618,E2 23260.618} C_VEL
LIN {X 0,Y 575.39,Z 806.236,A -85,B 0,C 180,E1 23259.938,E2 23259.938} C_VEL
LIN {X 0,Y 577.245,Z 764.459,A -85,B 0,C 180,E1 23259.303,E2 23259.303} C_VEL
LIN {X 0,Y 579.585,Z 714.399,A -85,B 0,C 180,E1 23258.606,E2 23258.606} C_VEL
LIN {X 0,Y 585.134,Z 660.022,A -85,B 0,C 180,E1 23257.688,E2 23257.688} C_VEL
LIN {X 0,Y 589.594,Z 616.706,A -85,B 0,C 180,E1 23256.961,E2 23256.961} C_VEL
LIN {X 0,Y 591.719,Z 598.474,A -85,B 0,C 180,E1 23256.686,E2 23256.686} C_VEL
LIN {X 0,Y 594.871,Z 567.651,A -85,B 0,C 180,E1 23256.166,E2 23256.166} C_VEL
LIN {X 0,Y 598.293,Z 540.605,A -85,B 0,C 180,E1 23255.791,E2 23255.791} C_VEL
LIN {X 0,Y 601.076,Z 512.789,A -85,B 0,C 180,E1 23255.315,E2 23255.315} C_VEL
LIN {X 0,Y 605.704,Z 478.07,A -85,B 0,C 180,E1 23254.865,E2 23254.865} C_VEL
LIN {X 0,Y 606.625,Z 466.298,A -85,B 0,C 180,E1 23254.631,E2 23254.631} C_VEL
LIN {X 0,Y 592.4,Z 443.36,A -85,B 0,C 180,E1 23252.005,E2 23252.005} C_VEL
LIN {X 0,Y 580.715,Z 425.719,A -85,B 0,C 180,E1 23249.643,E2 23249.643} C_VEL
LIN {X 0,Y 570.121,Z 410.612,A -85,B 0,C 180,E1 23247.299,E2 23247.299} C_VEL
LIN {X 0,Y 561.695,Z 399.302,A -85,B 0,C 180,E1 23245.264,E2 23245.264} C_VEL
LIN {X 0,Y 557.738,Z 394.056,A -85,B 0,C 180,E1 23244.239,E2 23244.239} C_VEL
LIN {X 0,Y 554.011,Z 389.148,A -85,B 0,C 180,E1 23243.226,E2 23243.226} C_VEL
LIN {X 0,Y 549.903,Z 383.902,A -85,B 0,C 180,E1 23242.054,E2 23242.054} C_VEL
LIN {X 0,Y 546.304,Z 379.312,A -85,B 0,C 180,E1 23240.966,E2 23240.966} C_VEL
LIN {X 0,Y 541.915,Z 374.017,A -85,B 0,C 180,E1 23239.566,E2 23239.566} C_VEL
LIN {X 0,Y 540.747,Z 372.36,A -85,B 0,C 180,E1 23239.161,E2 23239.161} C_VEL
LIN {X 0,Y 537.404,Z 368.833,A -85,B 0,C 180,E1 23238.019,E2 23238.019} C_VEL
LIN {X 0,Y 536.056,Z 366.422,A -85,B 0,C 180,E1 23237.476,E2 23237.476} C_VEL
LIN {X 0,Y 534.67,Z 365.613,A -85,B 0,C 180,E1 23237.004,E2 23237.004} C_VEL
LIN {X 0,Y 532.381,Z 369.548,A -85,B 0,C 180,E1 23236.531,E2 23236.531} C_VEL
LIN {X 0,Y 531.605,Z 370.724,A -85,B 0,C 180,E1 23236.358,E2 23236.358} C_VEL
LIN {X 0,Y 527.68,Z 382.688,A -85,B 0,C 180,E1 23235.849,E2 23235.849} C_VEL
LIN {X 0,Y 524.956,Z 389.498,A -85,B 0,C 180,E1 23235.381,E2 23235.381} C_VEL
LIN {X 0,Y 523.602,Z 392.135,A -85,B 0,C 180,E1 23235.053,E2 23235.053} C_VEL
LIN {X 0,Y 523.093,Z 478.801,A -85,B 0,C 180,E1 23231.774,E2 23231.774} C_VEL
LIN {X 0,Y 522.829,Z 551.62,A -85,B 0,C 180,E1 23228.912,E2 23228.912} C_VEL
LIN {X 0,Y 522.163,Z 626.715,A -85,B 0,C 180,E1 23225.88,E2 23225.88} C_VEL
LIN {X 0,Y 520.948,Z 712.014,A -85,B 0,C 180,E1 23222.365,E2 23222.365} C_VEL
LIN {X 0,Y 519.627,Z 790.172,A -85,B 0,C 180,E1 23219.063,E2 23219.063} C_VEL
LIN {X 0,Y 518.37,Z 852.348,A -85,B 0,C 180,E1 23216.406,E2 23216.406} C_VEL
LIN {X 0,Y 517.3,Z 866.567,A -85,B 0,C 180,E1 23215.846,E2 23215.846} C_VEL
LIN {X 0,Y 516.245,Z 974.401,A -85,B 0,C 180,E1 23214.197,E2 23214.197} C_VEL
LIN {X 0,Y 516.335,Z 990.627,A -85,B 0,C 180,E1 23213.816,E2 23213.816} C_VEL
LIN {X 0,Y 516.299,Z 1002.451,A -85,B 0,C 180,E1 23213.383,E2 23213.383} C_VEL
LIN {X 0,Y 516.159,Z 1013.904,A -85,B 0,C 180,E1 23212.822,E2 23212.822} C_VEL
LIN {X 0,Y 515.919,Z 1026.271,A -85,B 0,C 180,E1 23212.039,E2 23212.039} C_VEL
LIN {X 0,Y 515.575,Z 1037.813,A -85,B 0,C 180,E1 23211.074,E2 23211.074} C_VEL
LIN {X 0,Y 515.249,Z 1046.545,A -85,B 0,C 180,E1 23210.167,E2 23210.167} C_VEL
LIN {X 0,Y 514.946,Z 1053.79,A -85,B 0,C 180,E1 23209.257,E2 23209.257} C_VEL
LIN {X 0,Y 514.64,Z 1060.518,A -85,B 0,C 180,E1 23208.229,E2 23208.229} C_VEL
LIN {X 0,Y 514.369,Z 1066.011,A -85,B 0,C 180,E1 23207.197,E2 23207.197} C_VEL
LIN {X 0,Y 514.122,Z 1070.871,A -85,B 0,C 180,E1 23206.045,E2 23206.045} C_VEL
LIN {X 0,Y 513.914,Z 1074.896,A -85,B 0,C 180,E1 23204.772,E2 23204.772} C_VEL
LIN {X 0,Y 513.741,Z 1078.083,A -85,B 0,C 180,E1 23203.253,E2 23203.253} C_VEL
LIN {X 0,Y 513.635,Z 1079.423,A -85,B 0,C 180,E1 23201.735,E2 23201.735} C_VEL
LIN {X 0,Y 513.6,Z 1079.326,A -85,B 0,C 180,E1 23200.436,E2 23200.436} C_VEL
LIN {X 0,Y 513.617,Z 1078.044,A -85,B 0,C 180,E1 23199.129,E2 23199.129} C_VEL
LIN {X 0,Y 513.69,Z 1075.547,A -85,B 0,C 180,E1 23197.814,E2 23197.814} C_VEL
LIN {X 0,Y 513.852,Z 1071.373,A -85,B 0,C 180,E1 23196.369,E2 23196.369} C_VEL
LIN {X 0,Y 514.104,Z 1065.326,A -85,B 0,C 180,E1 23194.913,E2 23194.913} C_VEL
LIN {X 0,Y 514.393,Z 1058.429,A -85,B 0,C 180,E1 23193.652,E2 23193.652} C_VEL
LIN {X 0,Y 514.704,Z 1051.216,A -85,B 0,C 180,E1 23192.586,E2 23192.586} C_VEL
LIN {X 0,Y 515.082,Z 1042.003,A -85,B 0,C 180,E1 23191.475,E2 23191.475} C_VEL
LIN {X 0,Y 515.529,Z 1029.496,A -85,B 0,C 180,E1 23190.294,E2 23190.294} C_VEL
LIN {X 0,Y 515.838,Z 1018.487,A -85,B 0,C 180,E1 23189.479,E2 23189.479} C_VEL
LIN {X 0,Y 516.104,Z 1007.249,A -85,B 0,C 180,E1 23188.814,E2 23188.814} C_VEL
LIN {X 0,Y 516.329,Z 992.679,A -85,B 0,C 180,E1 23188.161,E2 23188.161} C_VEL
LIN {X 0,Y 516.364,Z 978.314,A -85,B 0,C 180,E1 23187.741,E2 23187.741} C_VEL
LIN {X 0,Y 516.313,Z 960.657,A -85,B 0,C 180,E1 23187.431,E2 23187.431} C_VEL
LIN {X 0,Y 517.529,Z 858.377,A -85,B 0,C 180,E1 23185.89,E2 23185.89} C_VEL
LIN {X 0,Y 518.446,Z 842.284,A -85,B 0,C 180,E1 23185.189,E2 23185.189} C_VEL
LIN {X 0,Y 519.126,Z 814.305,A -85,B 0,C 180,E1 23183.906,E2 23183.906} C_VEL
LIN {X 0,Y 520.218,Z 815.494,A -85,B 0,C 180,E1 23183.701,E2 23183.701} C_VEL
LIN {X 0,Y 522.172,Z 814.89,A -85,B 0,C 180,E1 23183.45,E2 23183.45} C_VEL
LIN {X 0,Y 525.115,Z 811.67,A -85,B 0,C 180,E1 23183.161,E2 23183.161} C_VEL
LIN {X 0,Y 528.611,Z 806.166,A -85,B 0,C 180,E1 23182.886,E2 23182.886} C_VEL
LIN {X 0,Y 531.848,Z 804.474,A -85,B 0,C 180,E1 23182.509,E2 23182.509} C_VEL
LIN {X 0,Y 535.612,Z 800.54,A -85,B 0,C 180,E1 23182.155,E2 23182.155} C_VEL
LIN {X 0,Y 538.772,Z 795.962,A -85,B 0,C 180,E1 23181.904,E2 23181.904} C_VEL
LIN {X 0,Y 543.153,Z 792.831,A -85,B 0,C 180,E1 23181.454,E2 23181.454} C_VEL
LIN {X 0,Y 547.819,Z 787.4,A -85,B 0,C 180,E1 23181.056,E2 23181.056} C_VEL
LIN {X 0,Y 549.558,Z 785.17,A -85,B 0,C 180,E1 23180.917,E2 23180.917} C_VEL
LIN {X 0,Y 554.64,Z 780.982,A -85,B 0,C 180,E1 23180.444,E2 23180.444} C_VEL
LIN {X 0,Y 560.479,Z 774.18,A -85,B 0,C 180,E1 23179.974,E2 23179.974} C_VEL
LIN {X 0,Y 566.386,Z 768.977,A -85,B 0,C 180,E1 23179.467,E2 23179.467} C_VEL
LIN {X 0,Y 567.849,Z 767.46,A -85,B 0,C 180,E1 23179.348,E2 23179.348} C_VEL
LIN {X 0,Y 563.812,Z 821.096,A -85,B 0,C 180,E1 23178.275,E2 23178.275} C_VEL
LIN {X 0,Y 561.185,Z 848.428,A -85,B 0,C 180,E1 23177.537,E2 23177.537} C_VEL
LIN {X 0,Y 560.932,Z 850.786,A -85,B 0,C 180,E1 23177.463,E2 23177.463} C_VEL
LIN {X 0,Y 559.271,Z 858.231,A -85,B 0,C 180,E1 23177.319,E2 23177.319} C_VEL
LIN {X 0,Y 552.44,Z 878.19,A -85,B 0,C 180,E1 23177.037,E2 23177.037} C_VEL
